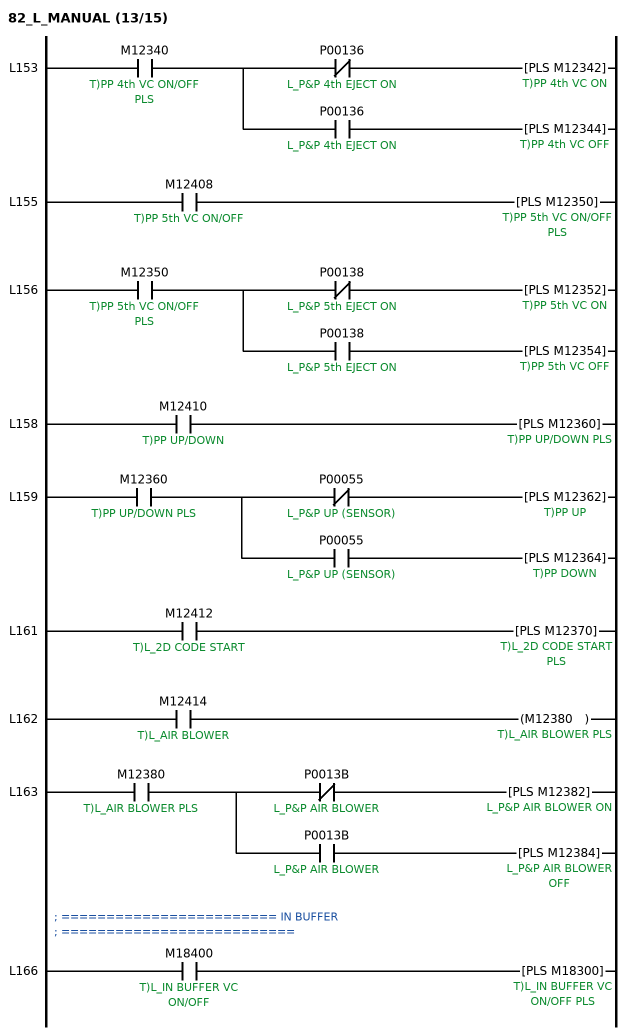
[picture p336: 82_L_MANUAL rungs L153-L166]
; L153
LOAD      M12340	// T)PP 4th VC ON/OFF PLS
MPUSH
AND NOT   P00136	// L_P&P 4th EJECT ON
OUTP      M12342	// T)PP 4th VC ON
MPOP
AND       P00136	// L_P&P 4th EJECT ON
OUTP      M12344	// T)PP 4th VC OFF
; L155
LOAD      M12408	// T)PP 5th VC ON/OFF
OUTP      M12350	// T)PP 5th VC ON/OFF PLS
; L156
LOAD      M12350	// T)PP 5th VC ON/OFF PLS
MPUSH
AND NOT   P00138	// L_P&P 5th EJECT ON
OUTP      M12352	// T)PP 5th VC ON
MPOP
AND       P00138	// L_P&P 5th EJECT ON
OUTP      M12354	// T)PP 5th VC OFF
; L158
LOAD      M12410	// T)PP UP/DOWN
OUTP      M12360	// T)PP UP/DOWN PLS
; L159
LOAD      M12360	// T)PP UP/DOWN PLS
MPUSH
AND NOT   P00055	// L_P&P UP (SENSOR)
OUTP      M12362	// T)PP UP
MPOP
AND       P00055	// L_P&P UP (SENSOR)
OUTP      M12364	// T)PP DOWN
; L161
LOAD      M12412	// T)L_2D CODE START
OUTP      M12370	// T)L_2D CODE START PLS
; L162
LOAD      M12414	// T)L_AIR BLOWER
OUT       M12380	// T)L_AIR BLOWER PLS
; L163
LOAD      M12380	// T)L_AIR BLOWER PLS
MPUSH
AND NOT   P0013B	// L_P&P AIR BLOWER
OUTP      M12382	// L_P&P AIR BLOWER ON
MPOP
AND       P0013B	// L_P&P AIR BLOWER
OUTP      M12384	// L_P&P AIR BLOWER OFF
// ======================== IN BUFFER ==========================
; L166
LOAD      M18400	// T)L_IN BUFFER VC ON/OFF
OUTP      M18300	// T)L_IN BUFFER VC ON/OFF PLS

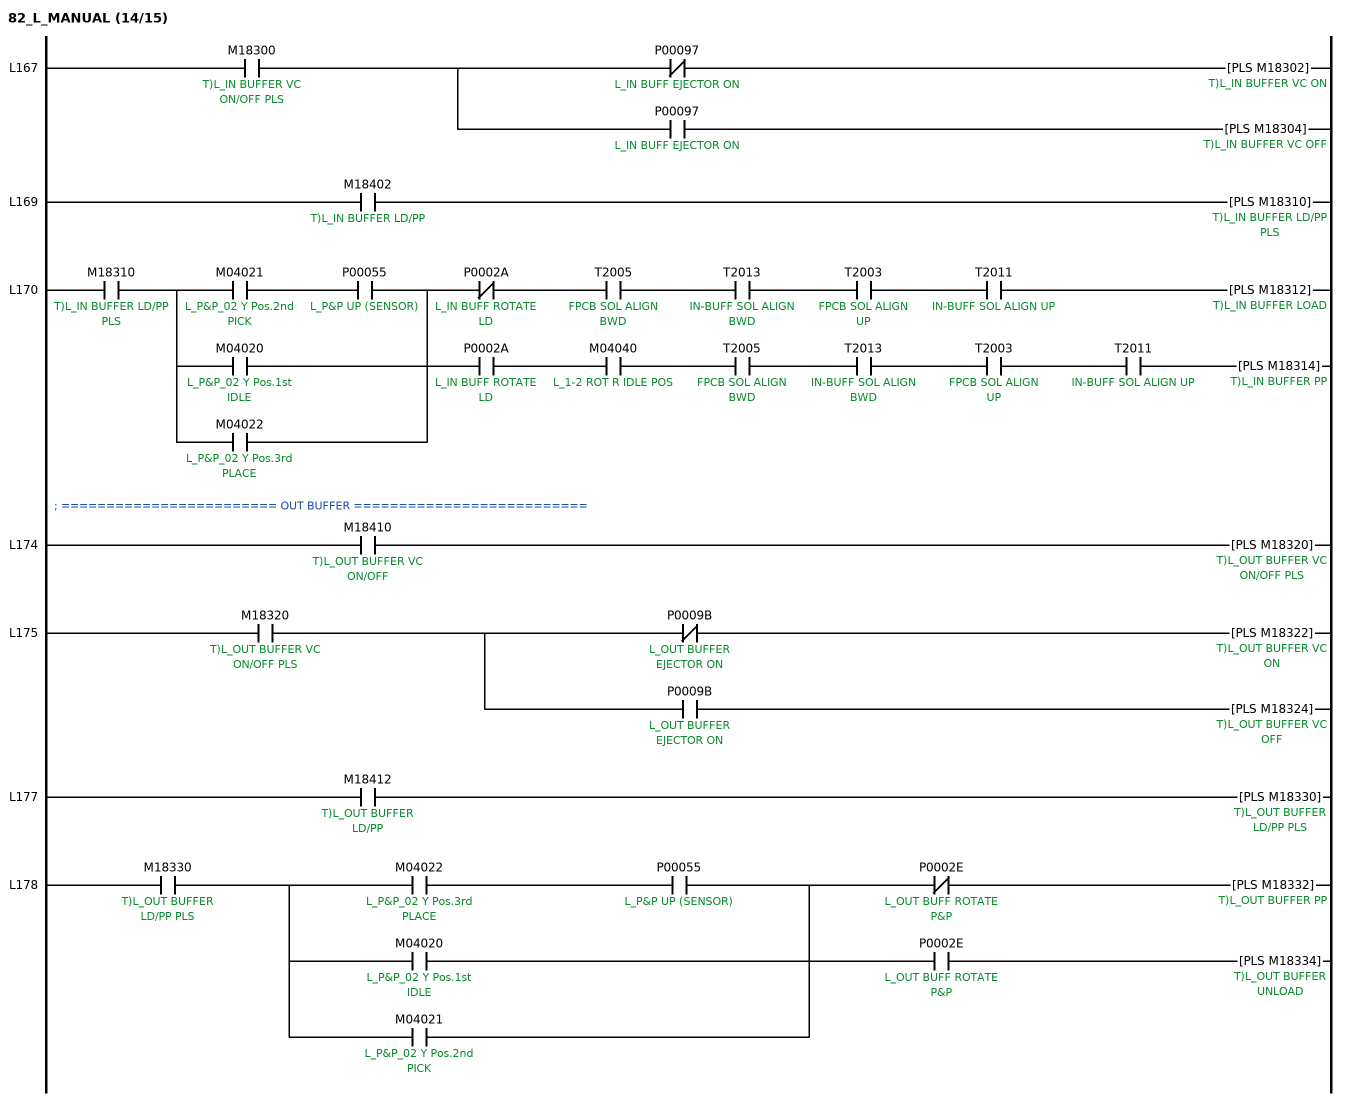
; L167
LOAD      M18300	// T)L_IN BUFFER VC ON/OFF PLS
MPUSH
AND NOT   P00097	// L_IN BUFF EJECTOR ON
OUTP      M18302	// T)L_IN BUFFER VC ON
MPOP
AND       P00097	// L_IN BUFF EJECTOR ON
OUTP      M18304	// T)L_IN BUFFER VC OFF
; L169
LOAD      M18402	// T)L_IN BUFFER LD/PP
OUTP      M18310	// T)L_IN BUFFER LD/PP PLS
; L170
LOAD      M18310	// T)L_IN BUFFER LD/PP PLS
LOAD      M04021	// L_P&P_02 Y Pos.2nd PICK
AND       P00055	// L_P&P UP (SENSOR)
OR        M04020	// L_P&P_02 Y Pos.1st IDLE
OR        M04022	// L_P&P_02 Y Pos.3rd PLACE
AND LOAD
MPUSH
AND NOT   P0002A	// L_IN BUFF ROTATE     LD
AND       T2005	// FPCB SOL ALIGN         BWD
AND       T2013	// IN-BUFF SOL ALIGN BWD
AND       T2003	// FPCB SOL ALIGN         UP
AND       T2011	// IN-BUFF SOL ALIGN UP
OUTP      M18312	// T)L_IN BUFFER LOAD
MPOP
AND       P0002A	// L_IN BUFF ROTATE     LD
AND       M04040	// L_1-2 ROT R IDLE POS
AND       T2005	// FPCB SOL ALIGN         BWD
AND       T2013	// IN-BUFF SOL ALIGN BWD
AND       T2003	// FPCB SOL ALIGN         UP
AND       T2011	// IN-BUFF SOL ALIGN UP
OUTP      M18314	// T)L_IN BUFFER PP
// ======================== OUT BUFFER ==========================
; L174
LOAD      M18410	// T)L_OUT BUFFER VC ON/OFF
OUTP      M18320	// T)L_OUT BUFFER VC ON/OFF PLS
; L175
LOAD      M18320	// T)L_OUT BUFFER VC ON/OFF PLS
MPUSH
AND NOT   P0009B	// L_OUT BUFFER EJECTOR ON
OUTP      M18322	// T)L_OUT BUFFER VC ON
MPOP
AND       P0009B	// L_OUT BUFFER EJECTOR ON
OUTP      M18324	// T)L_OUT BUFFER VC OFF
; L177
LOAD      M18412	// T)L_OUT BUFFER LD/PP
OUTP      M18330	// T)L_OUT BUFFER LD/PP PLS
; L178
LOAD      M18330	// T)L_OUT BUFFER LD/PP PLS
LOAD      M04022	// L_P&P_02 Y Pos.3rd PLACE
AND       P00055	// L_P&P UP (SENSOR)
OR        M04020	// L_P&P_02 Y Pos.1st IDLE
OR        M04021	// L_P&P_02 Y Pos.2nd PICK
AND LOAD
MPUSH
AND NOT   P0002E	// L_OUT BUFF ROTATE      P&P
OUTP      M18332	// T)L_OUT BUFFER PP
MPOP
AND       P0002E	// L_OUT BUFF ROTATE      P&P
OUTP      M18334	// T)L_OUT BUFFER UNLOAD

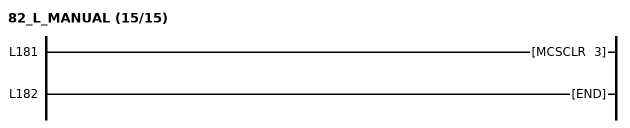
; L181
MCSCLR    3
; L182
END

PROGRAM 83_R_MANUAL (task: ¨ö¨¬A¥ì CA¡¤I¡¾¡¿¡¤¡Í)

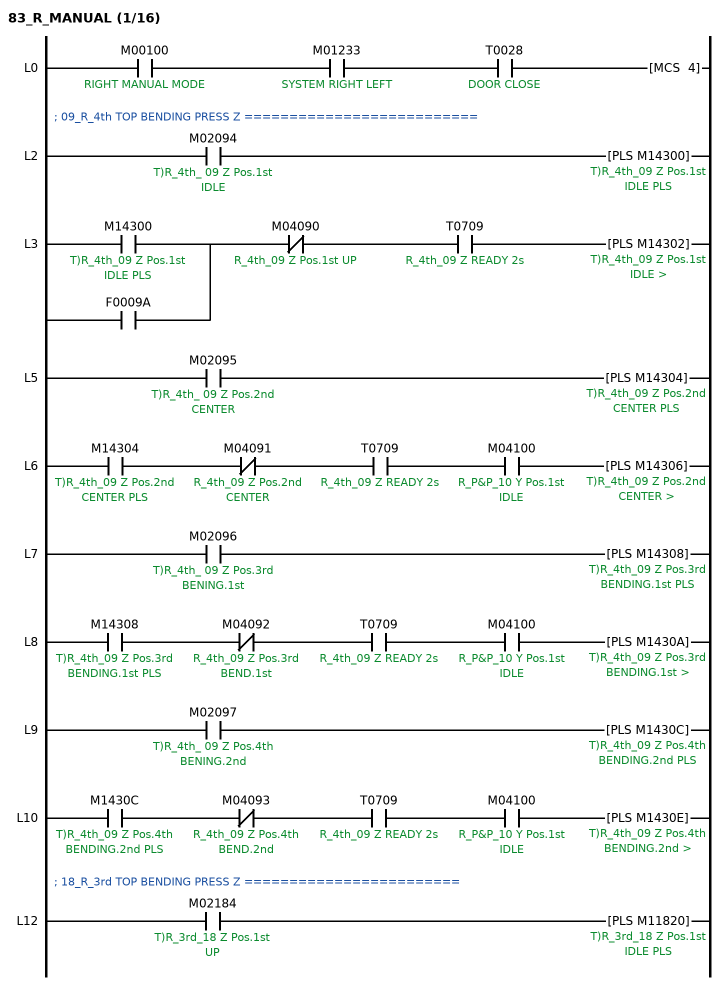
; L0
LOAD      M00100	// RIGHT MANUAL MODE
AND       M01233	// SYSTEM RIGHT LEFT
AND       T0028	// DOOR CLOSE
MCS       4
// 09_R_4th TOP BENDING PRESS Z ==========================
; L2
LOAD      M02094	// T)R_4th_ 09 Z Pos.1st IDLE
OUTP      M14300	// T)R_4th_09 Z Pos.1st IDLE PLS
; L3
LOAD      M14300	// T)R_4th_09 Z Pos.1st IDLE PLS
OR        F0009A
AND NOT   M04090	// R_4th_09 Z Pos.1st UP
AND       T0709	// R_4th_09 Z READY 2s
OUTP      M14302	// T)R_4th_09 Z Pos.1st IDLE >
; L5
LOAD      M02095	// T)R_4th_ 09 Z Pos.2nd CENTER
OUTP      M14304	// T)R_4th_09 Z Pos.2nd CENTER PLS
; L6
LOAD      M14304	// T)R_4th_09 Z Pos.2nd CENTER PLS
AND NOT   M04091	// R_4th_09 Z Pos.2nd CENTER
AND       T0709	// R_4th_09 Z READY 2s
AND       M04100	// R_P&P_10 Y Pos.1st IDLE
OUTP      M14306	// T)R_4th_09 Z Pos.2nd CENTER >
; L7
LOAD      M02096	// T)R_4th_ 09 Z Pos.3rd BENING.1st
OUTP      M14308	// T)R_4th_09 Z Pos.3rd BENDING.1st PLS
; L8
LOAD      M14308	// T)R_4th_09 Z Pos.3rd BENDING.1st PLS
AND NOT   M04092	// R_4th_09 Z Pos.3rd BEND.1st
AND       T0709	// R_4th_09 Z READY 2s
AND       M04100	// R_P&P_10 Y Pos.1st IDLE
OUTP      M1430A	// T)R_4th_09 Z Pos.3rd BENDING.1st >
; L9
LOAD      M02097	// T)R_4th_ 09 Z Pos.4th BENING.2nd
OUTP      M1430C	// T)R_4th_09 Z Pos.4th BENDING.2nd PLS
; L10
LOAD      M1430C	// T)R_4th_09 Z Pos.4th BENDING.2nd PLS
AND NOT   M04093	// R_4th_09 Z Pos.4th BEND.2nd
AND       T0709	// R_4th_09 Z READY 2s
AND       M04100	// R_P&P_10 Y Pos.1st IDLE
OUTP      M1430E	// T)R_4th_09 Z Pos.4th BENDING.2nd >
// 18_R_3rd TOP BENDING PRESS Z ======================== 
; L12
LOAD      M02184	// T)R_3rd_18 Z Pos.1st UP
OUTP      M11820	// T)R_3rd_18 Z Pos.1st IDLE PLS

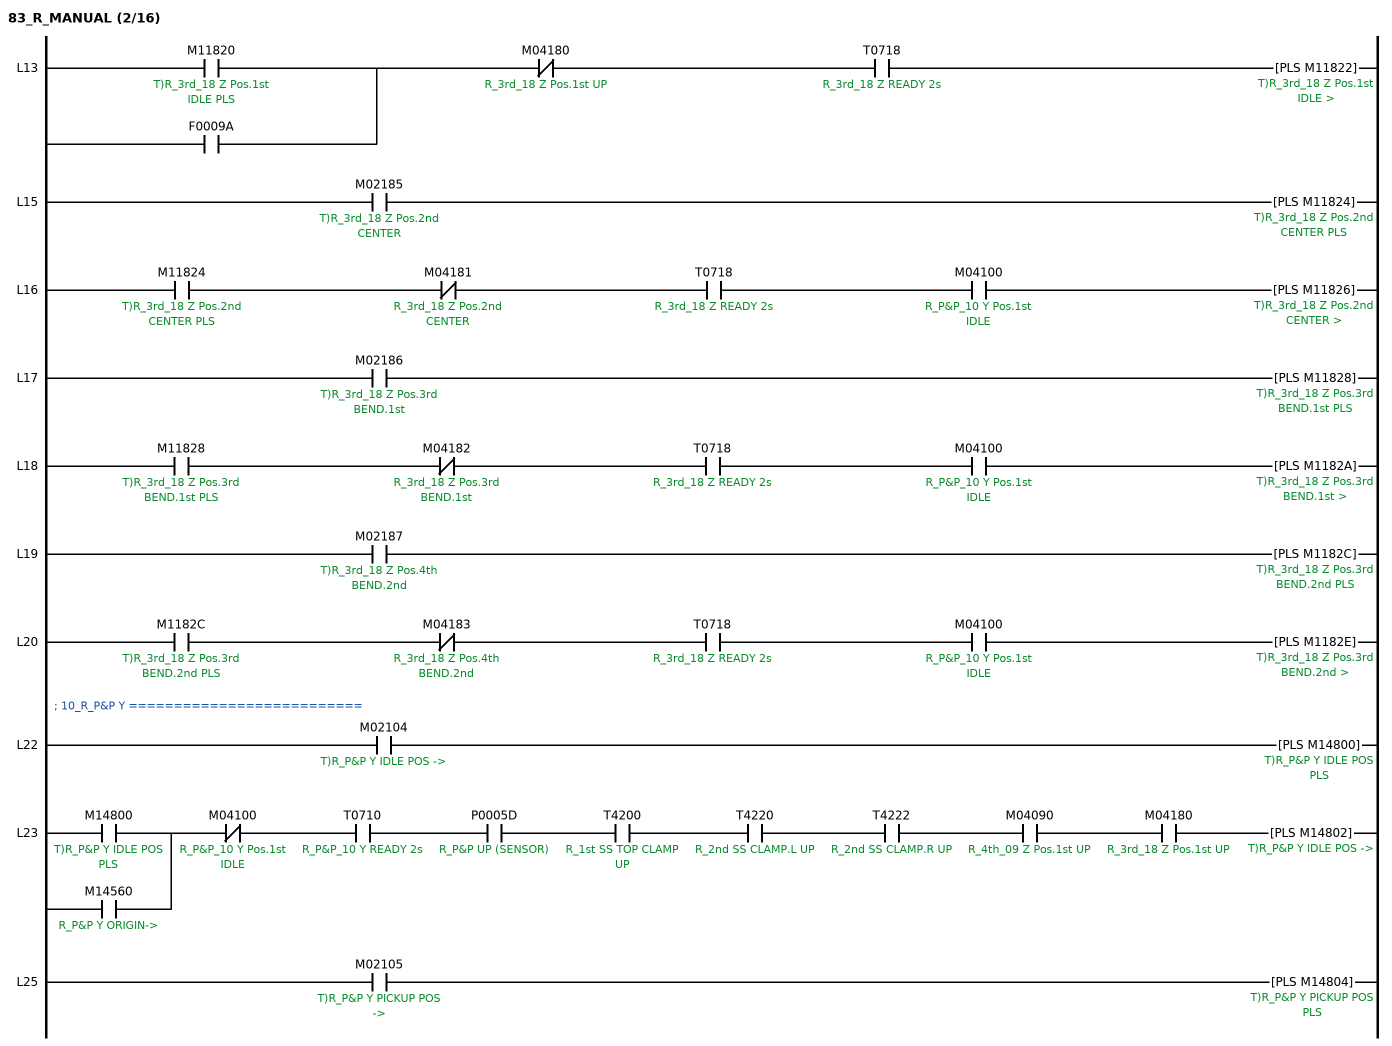
; L13
LOAD      M11820	// T)R_3rd_18 Z Pos.1st IDLE PLS
OR        F0009A
AND NOT   M04180	// R_3rd_18 Z Pos.1st UP
AND       T0718	// R_3rd_18 Z READY 2s
OUTP      M11822	// T)R_3rd_18 Z Pos.1st IDLE >
; L15
LOAD      M02185	// T)R_3rd_18 Z Pos.2nd CENTER
OUTP      M11824	// T)R_3rd_18 Z Pos.2nd CENTER PLS
; L16
LOAD      M11824	// T)R_3rd_18 Z Pos.2nd CENTER PLS
AND NOT   M04181	// R_3rd_18 Z Pos.2nd CENTER
AND       T0718	// R_3rd_18 Z READY 2s
AND       M04100	// R_P&P_10 Y Pos.1st IDLE
OUTP      M11826	// T)R_3rd_18 Z Pos.2nd CENTER >
; L17
LOAD      M02186	// T)R_3rd_18 Z Pos.3rd BEND.1st
OUTP      M11828	// T)R_3rd_18 Z Pos.3rd BEND.1st PLS
; L18
LOAD      M11828	// T)R_3rd_18 Z Pos.3rd BEND.1st PLS
AND NOT   M04182	// R_3rd_18 Z Pos.3rd BEND.1st
AND       T0718	// R_3rd_18 Z READY 2s
AND       M04100	// R_P&P_10 Y Pos.1st IDLE
OUTP      M1182A	// T)R_3rd_18 Z Pos.3rd BEND.1st >
; L19
LOAD      M02187	// T)R_3rd_18 Z Pos.4th BEND.2nd
OUTP      M1182C	// T)R_3rd_18 Z Pos.3rd BEND.2nd PLS
; L20
LOAD      M1182C	// T)R_3rd_18 Z Pos.3rd BEND.2nd PLS
AND NOT   M04183	// R_3rd_18 Z Pos.4th BEND.2nd
AND       T0718	// R_3rd_18 Z READY 2s
AND       M04100	// R_P&P_10 Y Pos.1st IDLE
OUTP      M1182E	// T)R_3rd_18 Z Pos.3rd BEND.2nd >
// 10_R_P&P Y ==========================
; L22
LOAD      M02104	// T)R_P&P Y IDLE POS ->
OUTP      M14800	// T)R_P&P Y IDLE POS PLS
; L23
LOAD      M14800	// T)R_P&P Y IDLE POS PLS
OR        M14560	// R_P&P Y ORIGIN->
AND NOT   M04100	// R_P&P_10 Y Pos.1st IDLE
AND       T0710	// R_P&P_10 Y READY 2s
AND       P0005D	// R_P&P UP (SENSOR)
AND       T4200	// R_1st SS TOP CLAMP UP
AND       T4220	// R_2nd SS CLAMP.L UP
AND       T4222	// R_2nd SS CLAMP.R UP
AND       M04090	// R_4th_09 Z Pos.1st UP
AND       M04180	// R_3rd_18 Z Pos.1st UP
OUTP      M14802	// T)R_P&P Y IDLE POS ->
; L25
LOAD      M02105	// T)R_P&P Y PICKUP POS ->
OUTP      M14804	// T)R_P&P Y PICKUP POS PLS

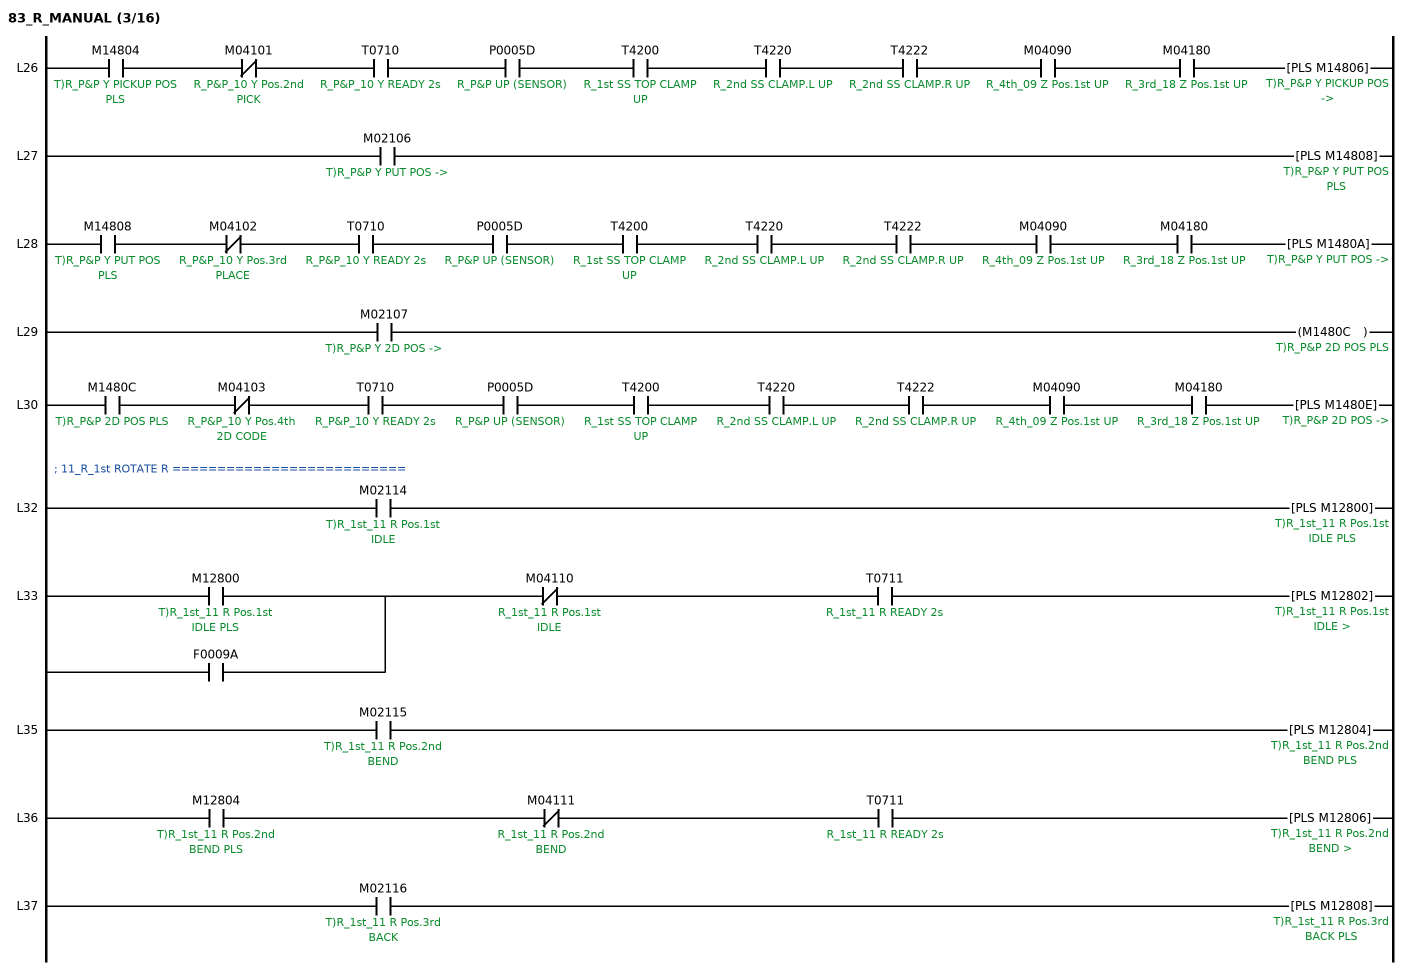
; L26
LOAD      M14804	// T)R_P&P Y PICKUP POS PLS
AND NOT   M04101	// R_P&P_10 Y Pos.2nd PICK
AND       T0710	// R_P&P_10 Y READY 2s
AND       P0005D	// R_P&P UP (SENSOR)
AND       T4200	// R_1st SS TOP CLAMP UP
AND       T4220	// R_2nd SS CLAMP.L UP
AND       T4222	// R_2nd SS CLAMP.R UP
AND       M04090	// R_4th_09 Z Pos.1st UP
AND       M04180	// R_3rd_18 Z Pos.1st UP
OUTP      M14806	// T)R_P&P Y PICKUP POS ->
; L27
LOAD      M02106	// T)R_P&P Y PUT POS ->
OUTP      M14808	// T)R_P&P Y PUT POS PLS
; L28
LOAD      M14808	// T)R_P&P Y PUT POS PLS
AND NOT   M04102	// R_P&P_10 Y Pos.3rd PLACE
AND       T0710	// R_P&P_10 Y READY 2s
AND       P0005D	// R_P&P UP (SENSOR)
AND       T4200	// R_1st SS TOP CLAMP UP
AND       T4220	// R_2nd SS CLAMP.L UP
AND       T4222	// R_2nd SS CLAMP.R UP
AND       M04090	// R_4th_09 Z Pos.1st UP
AND       M04180	// R_3rd_18 Z Pos.1st UP
OUTP      M1480A	// T)R_P&P Y PUT POS ->
; L29
LOAD      M02107	// T)R_P&P Y 2D POS ->
OUT       M1480C	// T)R_P&P 2D POS PLS
; L30
LOAD      M1480C	// T)R_P&P 2D POS PLS
AND NOT   M04103	// R_P&P_10 Y Pos.4th 2D CODE
AND       T0710	// R_P&P_10 Y READY 2s
AND       P0005D	// R_P&P UP (SENSOR)
AND       T4200	// R_1st SS TOP CLAMP UP
AND       T4220	// R_2nd SS CLAMP.L UP
AND       T4222	// R_2nd SS CLAMP.R UP
AND       M04090	// R_4th_09 Z Pos.1st UP
AND       M04180	// R_3rd_18 Z Pos.1st UP
OUTP      M1480E	// T)R_P&P 2D POS ->
// 11_R_1st ROTATE R ==========================
; L32
LOAD      M02114	// T)R_1st_11 R Pos.1st IDLE
OUTP      M12800	// T)R_1st_11 R Pos.1st IDLE PLS
; L33
LOAD      M12800	// T)R_1st_11 R Pos.1st IDLE PLS
OR        F0009A
AND NOT   M04110	// R_1st_11 R Pos.1st IDLE
AND       T0711	// R_1st_11 R READY 2s
OUTP      M12802	// T)R_1st_11 R Pos.1st IDLE >
; L35
LOAD      M02115	// T)R_1st_11 R Pos.2nd BEND
OUTP      M12804	// T)R_1st_11 R Pos.2nd BEND PLS
; L36
LOAD      M12804	// T)R_1st_11 R Pos.2nd BEND PLS
AND NOT   M04111	// R_1st_11 R Pos.2nd BEND
AND       T0711	// R_1st_11 R READY 2s
OUTP      M12806	// T)R_1st_11 R Pos.2nd BEND >
; L37
LOAD      M02116	// T)R_1st_11 R Pos.3rd BACK
OUTP      M12808	// T)R_1st_11 R Pos.3rd BACK PLS

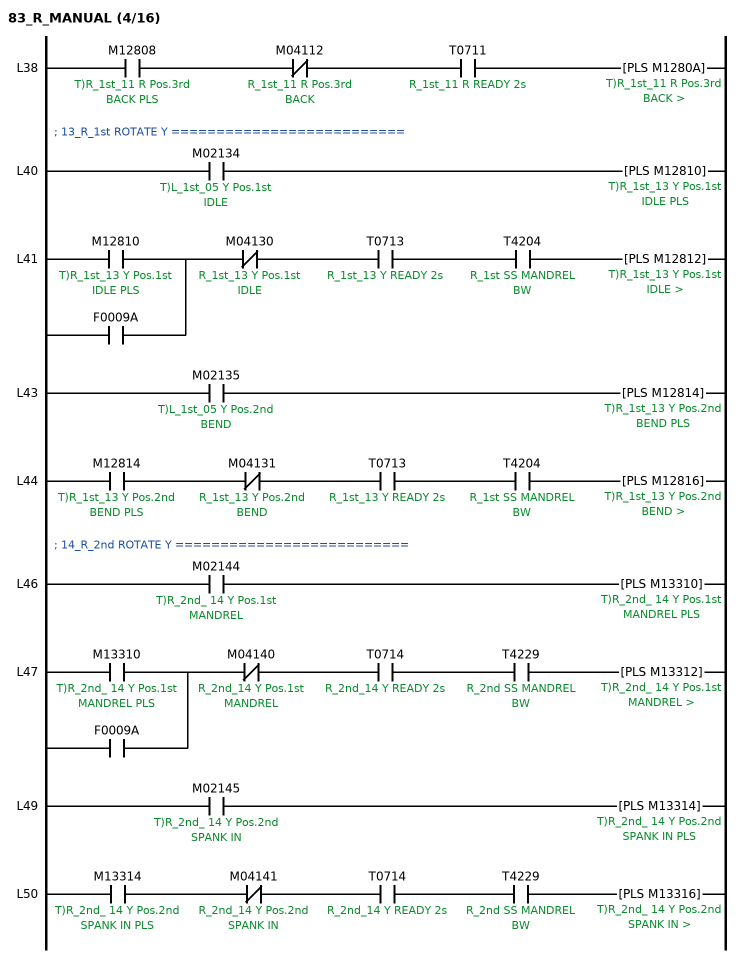
; L38
LOAD      M12808	// T)R_1st_11 R Pos.3rd BACK PLS
AND NOT   M04112	// R_1st_11 R Pos.3rd BACK
AND       T0711	// R_1st_11 R READY 2s
OUTP      M1280A	// T)R_1st_11 R Pos.3rd BACK >
// 13_R_1st ROTATE Y ==========================
; L40
LOAD      M02134	// T)L_1st_05 Y Pos.1st IDLE
OUTP      M12810	// T)R_1st_13 Y Pos.1st IDLE PLS
; L41
LOAD      M12810	// T)R_1st_13 Y Pos.1st IDLE PLS
OR        F0009A
AND NOT   M04130	// R_1st_13 Y Pos.1st IDLE
AND       T0713	// R_1st_13 Y READY 2s
AND       T4204	// R_1st SS MANDREL BW
OUTP      M12812	// T)R_1st_13 Y Pos.1st IDLE >
; L43
LOAD      M02135	// T)L_1st_05 Y Pos.2nd BEND
OUTP      M12814	// T)R_1st_13 Y Pos.2nd BEND PLS
; L44
LOAD      M12814	// T)R_1st_13 Y Pos.2nd BEND PLS
AND NOT   M04131	// R_1st_13 Y Pos.2nd BEND
AND       T0713	// R_1st_13 Y READY 2s
AND       T4204	// R_1st SS MANDREL BW
OUTP      M12816	// T)R_1st_13 Y Pos.2nd BEND >
// 14_R_2nd ROTATE Y ==========================
; L46
LOAD      M02144	// T)R_2nd_ 14 Y Pos.1st MANDREL
OUTP      M13310	// T)R_2nd_ 14 Y Pos.1st MANDREL PLS
; L47
LOAD      M13310	// T)R_2nd_ 14 Y Pos.1st MANDREL PLS
OR        F0009A
AND NOT   M04140	// R_2nd_14 Y Pos.1st MANDREL
AND       T0714	// R_2nd_14 Y READY 2s
AND       T4229	// R_2nd SS MANDREL BW
OUTP      M13312	// T)R_2nd_ 14 Y Pos.1st MANDREL >
; L49
LOAD      M02145	// T)R_2nd_ 14 Y Pos.2nd SPANK IN
OUTP      M13314	// T)R_2nd_ 14 Y Pos.2nd SPANK IN PLS
; L50
LOAD      M13314	// T)R_2nd_ 14 Y Pos.2nd SPANK IN PLS
AND NOT   M04141	// R_2nd_14 Y Pos.2nd SPANK IN
AND       T0714	// R_2nd_14 Y READY 2s
AND       T4229	// R_2nd SS MANDREL BW
OUTP      M13316	// T)R_2nd_ 14 Y Pos.2nd SPANK IN >

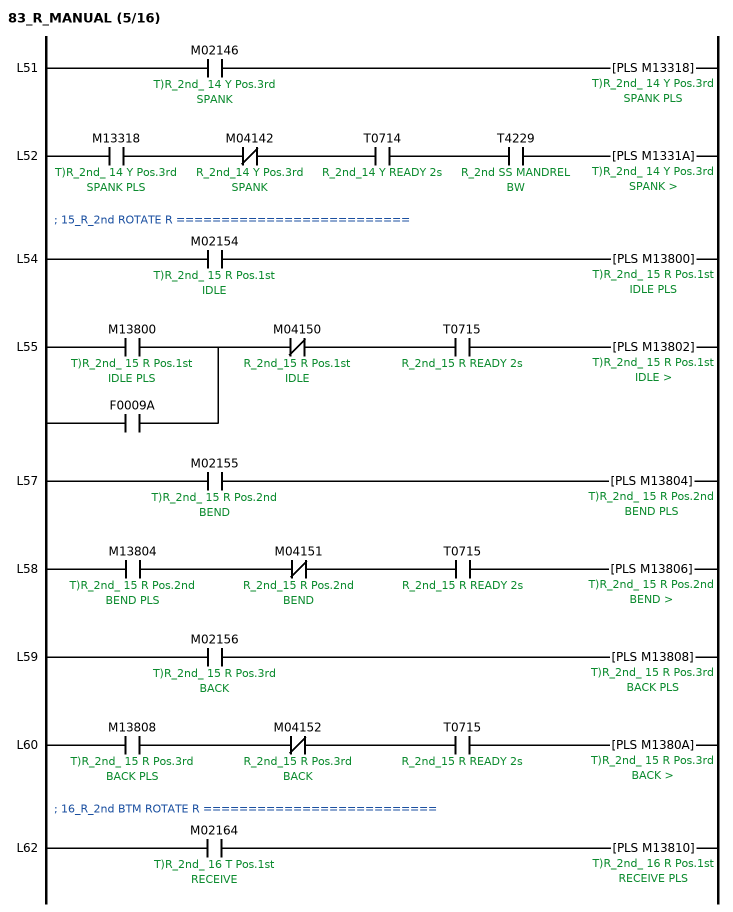
; L51
LOAD      M02146	// T)R_2nd_ 14 Y Pos.3rd SPANK
OUTP      M13318	// T)R_2nd_ 14 Y Pos.3rd SPANK PLS
; L52
LOAD      M13318	// T)R_2nd_ 14 Y Pos.3rd SPANK PLS
AND NOT   M04142	// R_2nd_14 Y Pos.3rd SPANK
AND       T0714	// R_2nd_14 Y READY 2s
AND       T4229	// R_2nd SS MANDREL BW
OUTP      M1331A	// T)R_2nd_ 14 Y Pos.3rd SPANK >
// 15_R_2nd ROTATE R ==========================
; L54
LOAD      M02154	// T)R_2nd_ 15 R Pos.1st IDLE
OUTP      M13800	// T)R_2nd_ 15 R Pos.1st IDLE PLS
; L55
LOAD      M13800	// T)R_2nd_ 15 R Pos.1st IDLE PLS
OR        F0009A
AND NOT   M04150	// R_2nd_15 R Pos.1st IDLE
AND       T0715	// R_2nd_15 R READY 2s
OUTP      M13802	// T)R_2nd_ 15 R Pos.1st IDLE >
; L57
LOAD      M02155	// T)R_2nd_ 15 R Pos.2nd BEND
OUTP      M13804	// T)R_2nd_ 15 R Pos.2nd BEND PLS
; L58
LOAD      M13804	// T)R_2nd_ 15 R Pos.2nd BEND PLS
AND NOT   M04151	// R_2nd_15 R Pos.2nd BEND
AND       T0715	// R_2nd_15 R READY 2s
OUTP      M13806	// T)R_2nd_ 15 R Pos.2nd BEND >
; L59
LOAD      M02156	// T)R_2nd_ 15 R Pos.3rd BACK
OUTP      M13808	// T)R_2nd_ 15 R Pos.3rd BACK PLS
; L60
LOAD      M13808	// T)R_2nd_ 15 R Pos.3rd BACK PLS
AND NOT   M04152	// R_2nd_15 R Pos.3rd BACK
AND       T0715	// R_2nd_15 R READY 2s
OUTP      M1380A	// T)R_2nd_ 15 R Pos.3rd BACK >
// 16_R_2nd BTM ROTATE R ==========================
; L62
LOAD      M02164	// T)R_2nd_ 16 T Pos.1st RECEIVE
OUTP      M13810	// T)R_2nd_ 16 R Pos.1st RECEIVE PLS

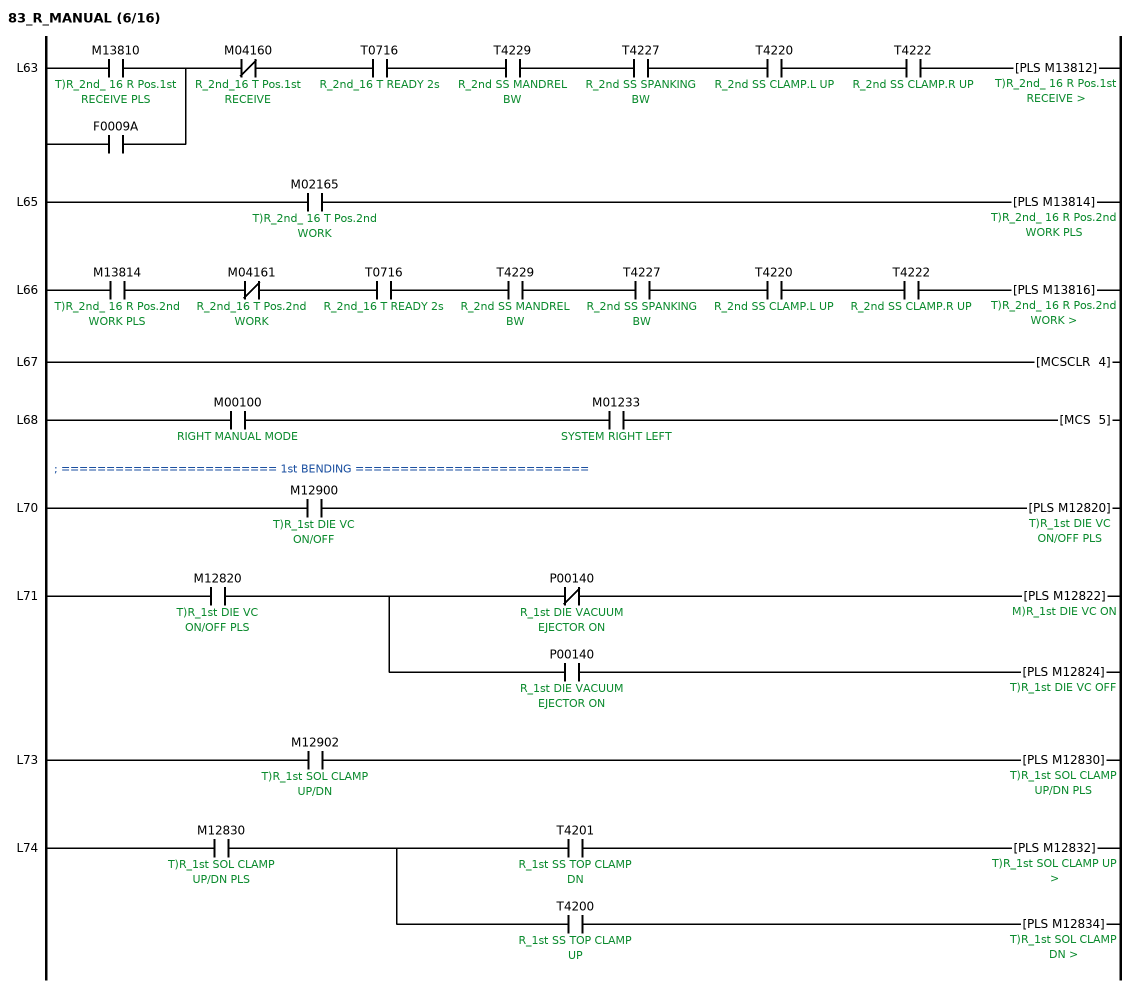
; L63
LOAD      M13810	// T)R_2nd_ 16 R Pos.1st RECEIVE PLS
OR        F0009A
AND NOT   M04160	// R_2nd_16 T Pos.1st RECEIVE
AND       T0716	// R_2nd_16 T READY 2s
AND       T4229	// R_2nd SS MANDREL BW
AND       T4227	// R_2nd SS SPANKING BW
AND       T4220	// R_2nd SS CLAMP.L UP
AND       T4222	// R_2nd SS CLAMP.R UP
OUTP      M13812	// T)R_2nd_ 16 R Pos.1st RECEIVE >
; L65
LOAD      M02165	// T)R_2nd_ 16 T Pos.2nd WORK
OUTP      M13814	// T)R_2nd_ 16 R Pos.2nd WORK PLS
; L66
LOAD      M13814	// T)R_2nd_ 16 R Pos.2nd WORK PLS
AND NOT   M04161	// R_2nd_16 T Pos.2nd WORK
AND       T0716	// R_2nd_16 T READY 2s
AND       T4229	// R_2nd SS MANDREL BW
AND       T4227	// R_2nd SS SPANKING BW
AND       T4220	// R_2nd SS CLAMP.L UP
AND       T4222	// R_2nd SS CLAMP.R UP
OUTP      M13816	// T)R_2nd_ 16 R Pos.2nd WORK >
; L67
MCSCLR    4
; L68
LOAD      M00100	// RIGHT MANUAL MODE
AND       M01233	// SYSTEM RIGHT LEFT
MCS       5
// ======================== 1st BENDING ==========================
; L70
LOAD      M12900	// T)R_1st DIE VC ON/OFF
OUTP      M12820	// T)R_1st DIE VC ON/OFF PLS
; L71
LOAD      M12820	// T)R_1st DIE VC ON/OFF PLS
MPUSH
AND NOT   P00140	// R_1st DIE VACUUM EJECTOR ON
OUTP      M12822	// M)R_1st DIE VC ON
MPOP
AND       P00140	// R_1st DIE VACUUM EJECTOR ON
OUTP      M12824	// T)R_1st DIE VC OFF
; L73
LOAD      M12902	// T)R_1st SOL CLAMP UP/DN
OUTP      M12830	// T)R_1st SOL CLAMP UP/DN PLS
; L74
LOAD      M12830	// T)R_1st SOL CLAMP UP/DN PLS
MPUSH
AND       T4201	// R_1st SS TOP CLAMP DN
OUTP      M12832	// T)R_1st SOL CLAMP UP >
MPOP
AND       T4200	// R_1st SS TOP CLAMP UP
OUTP      M12834	// T)R_1st SOL CLAMP DN >

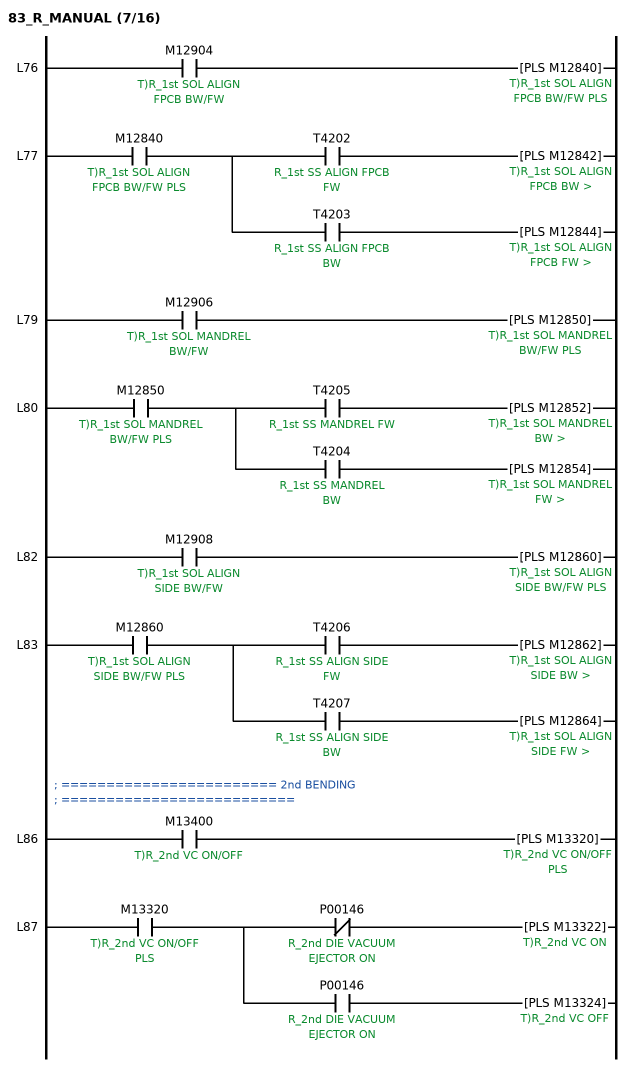
; L76
LOAD      M12904	// T)R_1st SOL ALIGN FPCB BW/FW
OUTP      M12840	// T)R_1st SOL ALIGN FPCB BW/FW PLS
; L77
LOAD      M12840	// T)R_1st SOL ALIGN FPCB BW/FW PLS
MPUSH
AND       T4202	// R_1st SS ALIGN FPCB FW
OUTP      M12842	// T)R_1st SOL ALIGN FPCB BW >
MPOP
AND       T4203	// R_1st SS ALIGN FPCB BW
OUTP      M12844	// T)R_1st SOL ALIGN FPCB FW >
; L79
LOAD      M12906	// T)R_1st SOL MANDREL BW/FW
OUTP      M12850	// T)R_1st SOL MANDREL BW/FW PLS
; L80
LOAD      M12850	// T)R_1st SOL MANDREL BW/FW PLS
MPUSH
AND       T4205	// R_1st SS MANDREL FW
OUTP      M12852	// T)R_1st SOL MANDREL BW >
MPOP
AND       T4204	// R_1st SS MANDREL BW
OUTP      M12854	// T)R_1st SOL MANDREL FW >
; L82
LOAD      M12908	// T)R_1st SOL ALIGN SIDE BW/FW
OUTP      M12860	// T)R_1st SOL ALIGN SIDE BW/FW PLS
; L83
LOAD      M12860	// T)R_1st SOL ALIGN SIDE BW/FW PLS
MPUSH
AND       T4206	// R_1st SS ALIGN SIDE FW
OUTP      M12862	// T)R_1st SOL ALIGN SIDE BW >
MPOP
AND       T4207	// R_1st SS ALIGN SIDE BW
OUTP      M12864	// T)R_1st SOL ALIGN SIDE FW >
// ======================== 2nd BENDING ==========================
; L86
LOAD      M13400	// T)R_2nd VC ON/OFF
OUTP      M13320	// T)R_2nd VC ON/OFF PLS
; L87
LOAD      M13320	// T)R_2nd VC ON/OFF PLS
MPUSH
AND NOT   P00146	// R_2nd DIE VACUUM EJECTOR ON
OUTP      M13322	// T)R_2nd VC ON
MPOP
AND       P00146	// R_2nd DIE VACUUM EJECTOR ON
OUTP      M13324	// T)R_2nd VC OFF

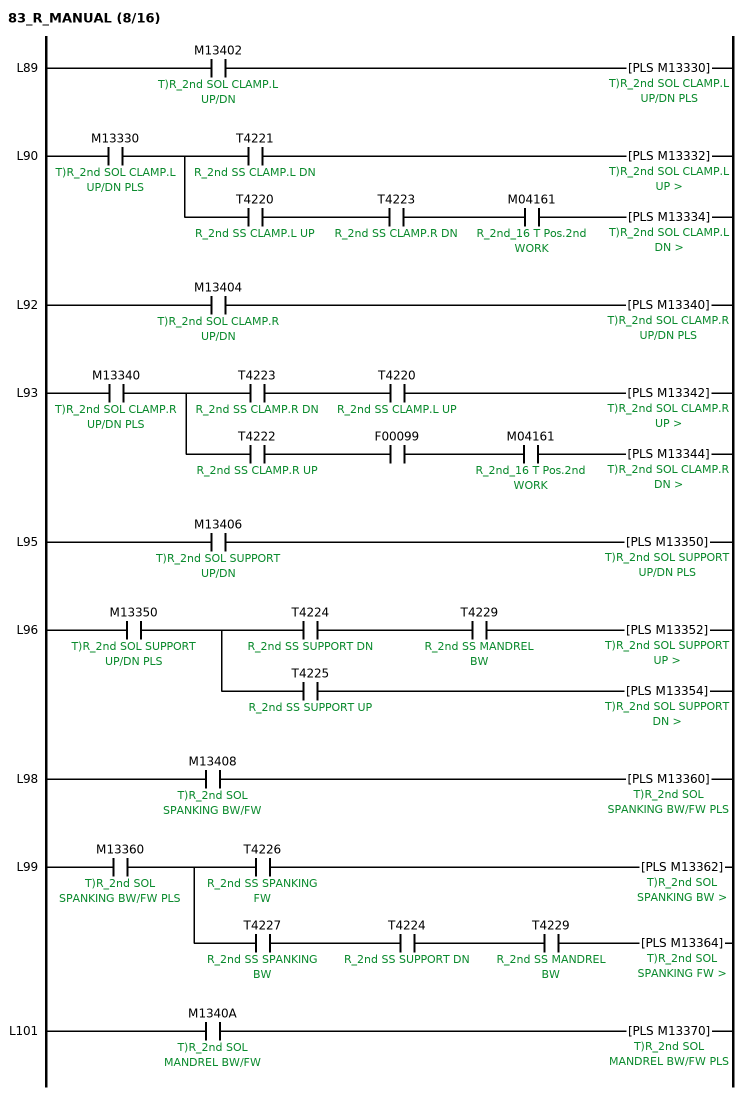
; L89
LOAD      M13402	// T)R_2nd SOL CLAMP.L UP/DN
OUTP      M13330	// T)R_2nd SOL CLAMP.L UP/DN PLS
; L90
LOAD      M13330	// T)R_2nd SOL CLAMP.L UP/DN PLS
MPUSH
AND       T4221	// R_2nd SS CLAMP.L DN
OUTP      M13332	// T)R_2nd SOL CLAMP.L UP >
MPOP
AND       T4220	// R_2nd SS CLAMP.L UP
AND       T4223	// R_2nd SS CLAMP.R DN
AND       M04161	// R_2nd_16 T Pos.2nd WORK
OUTP      M13334	// T)R_2nd SOL CLAMP.L DN >
; L92
LOAD      M13404	// T)R_2nd SOL CLAMP.R UP/DN
OUTP      M13340	// T)R_2nd SOL CLAMP.R UP/DN PLS
; L93
LOAD      M13340	// T)R_2nd SOL CLAMP.R UP/DN PLS
MPUSH
AND       T4223	// R_2nd SS CLAMP.R DN
AND       T4220	// R_2nd SS CLAMP.L UP
OUTP      M13342	// T)R_2nd SOL CLAMP.R UP >
MPOP
AND       T4222	// R_2nd SS CLAMP.R UP
AND       F00099
AND       M04161	// R_2nd_16 T Pos.2nd WORK
OUTP      M13344	// T)R_2nd SOL CLAMP.R DN >
; L95
LOAD      M13406	// T)R_2nd SOL SUPPORT UP/DN
OUTP      M13350	// T)R_2nd SOL SUPPORT UP/DN PLS
; L96
LOAD      M13350	// T)R_2nd SOL SUPPORT UP/DN PLS
MPUSH
AND       T4224	// R_2nd SS SUPPORT DN
AND       T4229	// R_2nd SS MANDREL BW
OUTP      M13352	// T)R_2nd SOL SUPPORT UP >
MPOP
AND       T4225	// R_2nd SS SUPPORT UP
OUTP      M13354	// T)R_2nd SOL SUPPORT DN >
; L98
LOAD      M13408	// T)R_2nd SOL SPANKING BW/FW
OUTP      M13360	// T)R_2nd SOL SPANKING BW/FW PLS
; L99
LOAD      M13360	// T)R_2nd SOL SPANKING BW/FW PLS
MPUSH
AND       T4226	// R_2nd SS SPANKING FW
OUTP      M13362	// T)R_2nd SOL SPANKING BW >
MPOP
AND       T4227	// R_2nd SS SPANKING BW
AND       T4224	// R_2nd SS SUPPORT DN
AND       T4229	// R_2nd SS MANDREL BW
OUTP      M13364	// T)R_2nd SOL SPANKING FW >
; L101
LOAD      M1340A	// T)R_2nd SOL MANDREL BW/FW
OUTP      M13370	// T)R_2nd SOL MANDREL BW/FW PLS

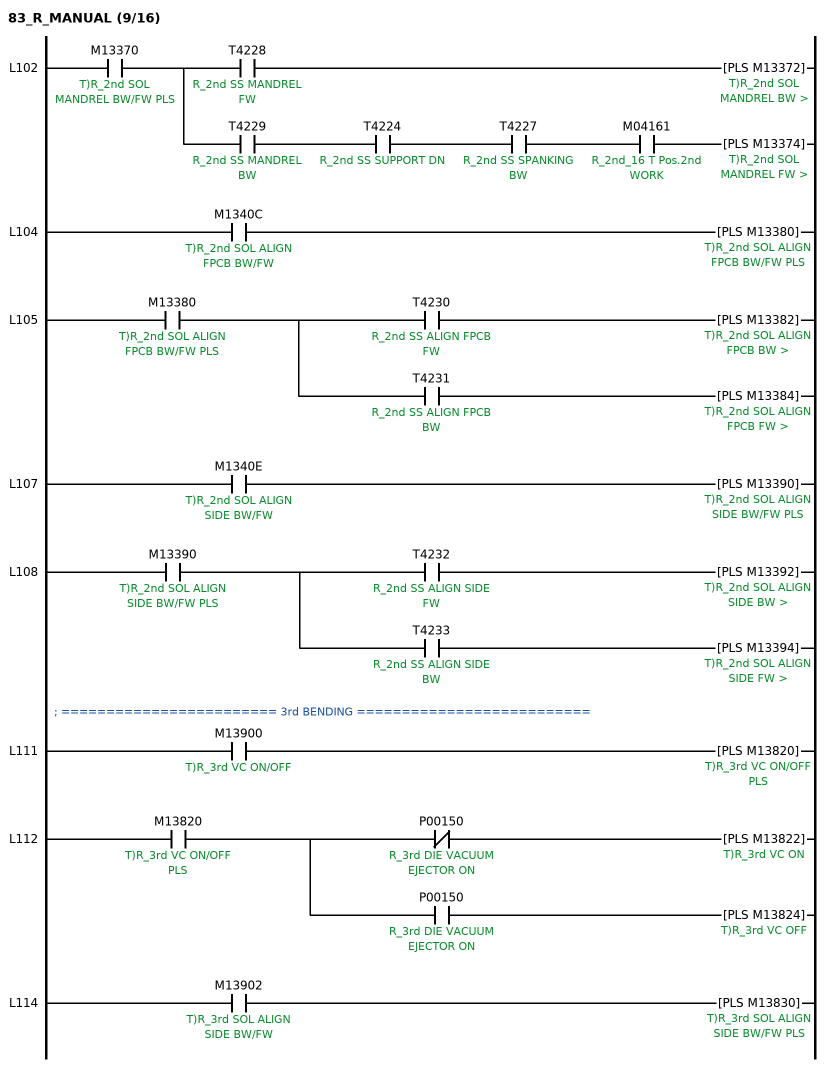
; L102
LOAD      M13370	// T)R_2nd SOL MANDREL BW/FW PLS
MPUSH
AND       T4228	// R_2nd SS MANDREL FW
OUTP      M13372	// T)R_2nd SOL MANDREL BW >
MPOP
AND       T4229	// R_2nd SS MANDREL BW
AND       T4224	// R_2nd SS SUPPORT DN
AND       T4227	// R_2nd SS SPANKING BW
AND       M04161	// R_2nd_16 T Pos.2nd WORK
OUTP      M13374	// T)R_2nd SOL MANDREL FW >
; L104
LOAD      M1340C	// T)R_2nd SOL ALIGN FPCB BW/FW
OUTP      M13380	// T)R_2nd SOL ALIGN FPCB BW/FW PLS
; L105
LOAD      M13380	// T)R_2nd SOL ALIGN FPCB BW/FW PLS
MPUSH
AND       T4230	// R_2nd SS ALIGN FPCB FW
OUTP      M13382	// T)R_2nd SOL ALIGN FPCB BW >
MPOP
AND       T4231	// R_2nd SS ALIGN FPCB BW
OUTP      M13384	// T)R_2nd SOL ALIGN FPCB FW >
; L107
LOAD      M1340E	// T)R_2nd SOL ALIGN SIDE BW/FW
OUTP      M13390	// T)R_2nd SOL ALIGN SIDE BW/FW PLS
; L108
LOAD      M13390	// T)R_2nd SOL ALIGN SIDE BW/FW PLS
MPUSH
AND       T4232	// R_2nd SS ALIGN SIDE FW
OUTP      M13392	// T)R_2nd SOL ALIGN SIDE BW >
MPOP
AND       T4233	// R_2nd SS ALIGN SIDE BW
OUTP      M13394	// T)R_2nd SOL ALIGN SIDE FW >
// ======================== 3rd BENDING ==========================
; L111
LOAD      M13900	// T)R_3rd VC ON/OFF
OUTP      M13820	// T)R_3rd VC ON/OFF PLS
; L112
LOAD      M13820	// T)R_3rd VC ON/OFF PLS
MPUSH
AND NOT   P00150	// R_3rd DIE VACUUM EJECTOR ON
OUTP      M13822	// T)R_3rd VC ON
MPOP
AND       P00150	// R_3rd DIE VACUUM EJECTOR ON
OUTP      M13824	// T)R_3rd VC OFF
; L114
LOAD      M13902	// T)R_3rd SOL ALIGN SIDE BW/FW
OUTP      M13830	// T)R_3rd SOL ALIGN SIDE BW/FW PLS

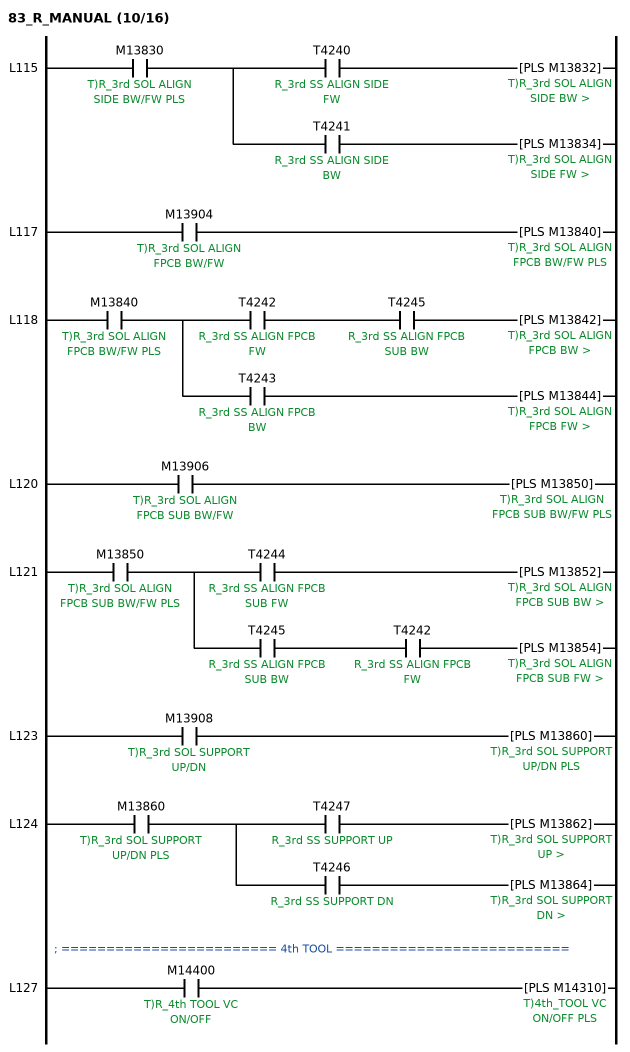
; L115
LOAD      M13830	// T)R_3rd SOL ALIGN SIDE BW/FW PLS
MPUSH
AND       T4240	// R_3rd SS ALIGN SIDE FW
OUTP      M13832	// T)R_3rd SOL ALIGN SIDE BW >
MPOP
AND       T4241	// R_3rd SS ALIGN SIDE BW
OUTP      M13834	// T)R_3rd SOL ALIGN SIDE FW >
; L117
LOAD      M13904	// T)R_3rd SOL ALIGN FPCB BW/FW
OUTP      M13840	// T)R_3rd SOL ALIGN FPCB BW/FW PLS
; L118
LOAD      M13840	// T)R_3rd SOL ALIGN FPCB BW/FW PLS
MPUSH
AND       T4242	// R_3rd SS ALIGN FPCB FW
AND       T4245	// R_3rd SS ALIGN FPCB SUB BW
OUTP      M13842	// T)R_3rd SOL ALIGN FPCB BW >
MPOP
AND       T4243	// R_3rd SS ALIGN FPCB BW
OUTP      M13844	// T)R_3rd SOL ALIGN FPCB FW >
; L120
LOAD      M13906	// T)R_3rd SOL ALIGN FPCB SUB BW/FW
OUTP      M13850	// T)R_3rd SOL ALIGN FPCB SUB BW/FW PLS
; L121
LOAD      M13850	// T)R_3rd SOL ALIGN FPCB SUB BW/FW PLS
MPUSH
AND       T4244	// R_3rd SS ALIGN FPCB SUB FW
OUTP      M13852	// T)R_3rd SOL ALIGN FPCB SUB BW >
MPOP
AND       T4245	// R_3rd SS ALIGN FPCB SUB BW
AND       T4242	// R_3rd SS ALIGN FPCB FW
OUTP      M13854	// T)R_3rd SOL ALIGN FPCB SUB FW >
; L123
LOAD      M13908	// T)R_3rd SOL SUPPORT UP/DN
OUTP      M13860	// T)R_3rd SOL SUPPORT UP/DN PLS
; L124
LOAD      M13860	// T)R_3rd SOL SUPPORT UP/DN PLS
MPUSH
AND       T4247	// R_3rd SS SUPPORT UP
OUTP      M13862	// T)R_3rd SOL SUPPORT UP >
MPOP
AND       T4246	// R_3rd SS SUPPORT DN
OUTP      M13864	// T)R_3rd SOL SUPPORT DN >
// ======================== 4th TOOL ==========================
; L127
LOAD      M14400	// T)R_4th TOOL VC ON/OFF
OUTP      M14310	// T)4th_TOOL VC ON/OFF PLS

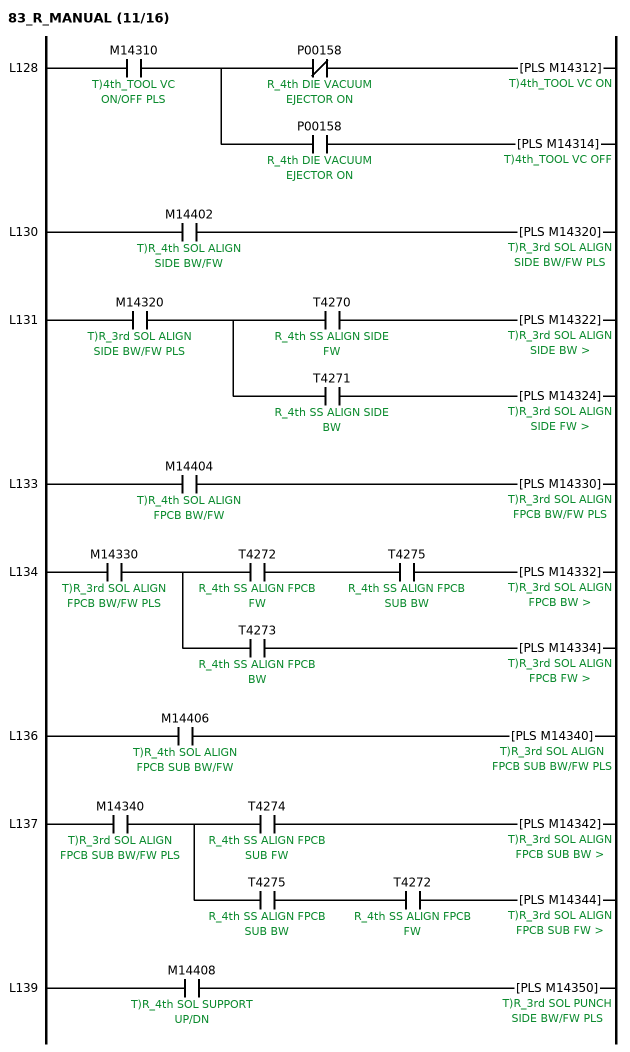
; L128
LOAD      M14310	// T)4th_TOOL VC ON/OFF PLS
MPUSH
AND NOT   P00158	// R_4th DIE VACUUM EJECTOR ON
OUTP      M14312	// T)4th_TOOL VC ON
MPOP
AND       P00158	// R_4th DIE VACUUM EJECTOR ON
OUTP      M14314	// T)4th_TOOL VC OFF
; L130
LOAD      M14402	// T)R_4th SOL ALIGN SIDE BW/FW
OUTP      M14320	// T)R_3rd SOL ALIGN SIDE BW/FW PLS
; L131
LOAD      M14320	// T)R_3rd SOL ALIGN SIDE BW/FW PLS
MPUSH
AND       T4270	// R_4th SS ALIGN SIDE FW
OUTP      M14322	// T)R_3rd SOL ALIGN SIDE BW >
MPOP
AND       T4271	// R_4th SS ALIGN SIDE BW
OUTP      M14324	// T)R_3rd SOL ALIGN SIDE FW >
; L133
LOAD      M14404	// T)R_4th SOL ALIGN FPCB BW/FW
OUTP      M14330	// T)R_3rd SOL ALIGN FPCB BW/FW PLS
; L134
LOAD      M14330	// T)R_3rd SOL ALIGN FPCB BW/FW PLS
MPUSH
AND       T4272	// R_4th SS ALIGN FPCB FW
AND       T4275	// R_4th SS ALIGN FPCB SUB BW
OUTP      M14332	// T)R_3rd SOL ALIGN FPCB BW >
MPOP
AND       T4273	// R_4th SS ALIGN FPCB BW
OUTP      M14334	// T)R_3rd SOL ALIGN FPCB FW >
; L136
LOAD      M14406	// T)R_4th SOL ALIGN FPCB SUB BW/FW
OUTP      M14340	// T)R_3rd SOL ALIGN FPCB SUB BW/FW PLS
; L137
LOAD      M14340	// T)R_3rd SOL ALIGN FPCB SUB BW/FW PLS
MPUSH
AND       T4274	// R_4th SS ALIGN FPCB SUB FW
OUTP      M14342	// T)R_3rd SOL ALIGN FPCB SUB BW >
MPOP
AND       T4275	// R_4th SS ALIGN FPCB SUB BW
AND       T4272	// R_4th SS ALIGN FPCB FW
OUTP      M14344	// T)R_3rd SOL ALIGN FPCB SUB FW >
; L139
LOAD      M14408	// T)R_4th SOL SUPPORT UP/DN
OUTP      M14350	// T)R_3rd SOL PUNCH SIDE BW/FW PLS

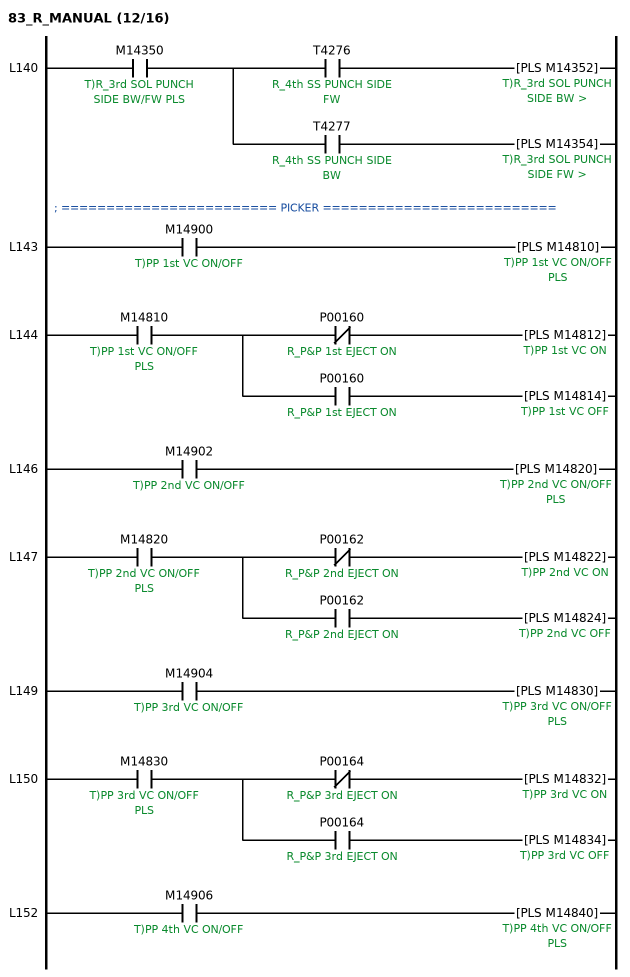
; L140
LOAD      M14350	// T)R_3rd SOL PUNCH SIDE BW/FW PLS
MPUSH
AND       T4276	// R_4th SS PUNCH SIDE FW
OUTP      M14352	// T)R_3rd SOL PUNCH SIDE BW >
MPOP
AND       T4277	// R_4th SS PUNCH SIDE BW
OUTP      M14354	// T)R_3rd SOL PUNCH SIDE FW >
// ======================== PICKER ==========================
; L143
LOAD      M14900	// T)PP 1st VC ON/OFF
OUTP      M14810	// T)PP 1st VC ON/OFF PLS
; L144
LOAD      M14810	// T)PP 1st VC ON/OFF PLS
MPUSH
AND NOT   P00160	// R_P&P 1st EJECT ON
OUTP      M14812	// T)PP 1st VC ON
MPOP
AND       P00160	// R_P&P 1st EJECT ON
OUTP      M14814	// T)PP 1st VC OFF
; L146
LOAD      M14902	// T)PP 2nd VC ON/OFF
OUTP      M14820	// T)PP 2nd VC ON/OFF PLS
; L147
LOAD      M14820	// T)PP 2nd VC ON/OFF PLS
MPUSH
AND NOT   P00162	// R_P&P 2nd EJECT ON
OUTP      M14822	// T)PP 2nd VC ON
MPOP
AND       P00162	// R_P&P 2nd EJECT ON
OUTP      M14824	// T)PP 2nd VC OFF
; L149
LOAD      M14904	// T)PP 3rd VC ON/OFF
OUTP      M14830	// T)PP 3rd VC ON/OFF PLS
; L150
LOAD      M14830	// T)PP 3rd VC ON/OFF PLS
MPUSH
AND NOT   P00164	// R_P&P 3rd EJECT ON
OUTP      M14832	// T)PP 3rd VC ON
MPOP
AND       P00164	// R_P&P 3rd EJECT ON
OUTP      M14834	// T)PP 3rd VC OFF
; L152
LOAD      M14906	// T)PP 4th VC ON/OFF
OUTP      M14840	// T)PP 4th VC ON/OFF PLS

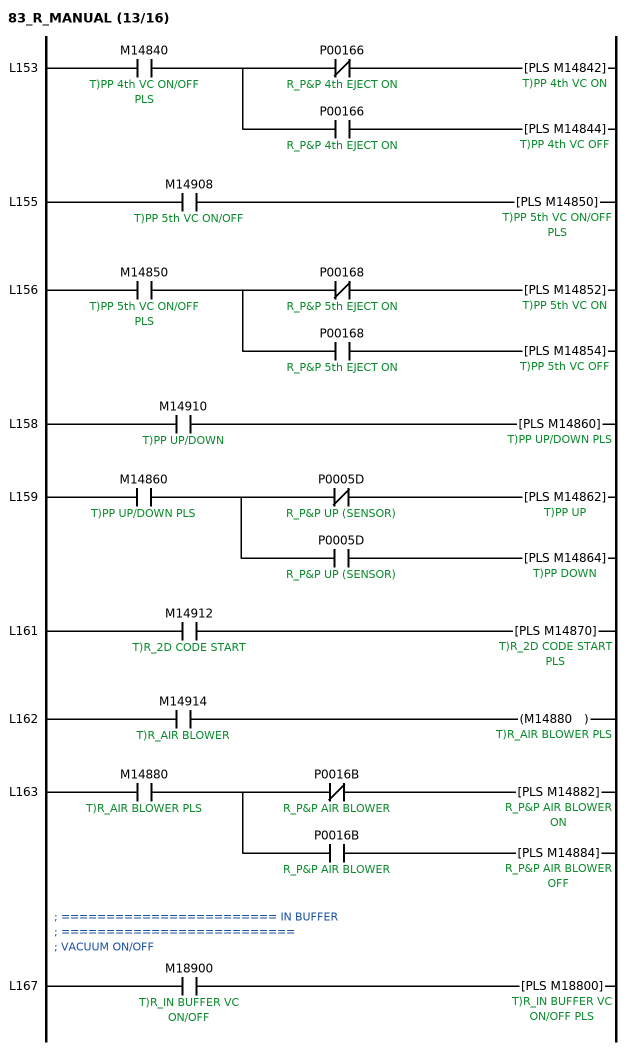
; L153
LOAD      M14840	// T)PP 4th VC ON/OFF PLS
MPUSH
AND NOT   P00166	// R_P&P 4th EJECT ON
OUTP      M14842	// T)PP 4th VC ON
MPOP
AND       P00166	// R_P&P 4th EJECT ON
OUTP      M14844	// T)PP 4th VC OFF
; L155
LOAD      M14908	// T)PP 5th VC ON/OFF
OUTP      M14850	// T)PP 5th VC ON/OFF PLS
; L156
LOAD      M14850	// T)PP 5th VC ON/OFF PLS
MPUSH
AND NOT   P00168	// R_P&P 5th EJECT ON
OUTP      M14852	// T)PP 5th VC ON
MPOP
AND       P00168	// R_P&P 5th EJECT ON
OUTP      M14854	// T)PP 5th VC OFF
; L158
LOAD      M14910	// T)PP UP/DOWN
OUTP      M14860	// T)PP UP/DOWN PLS
; L159
LOAD      M14860	// T)PP UP/DOWN PLS
MPUSH
AND NOT   P0005D	// R_P&P UP (SENSOR)
OUTP      M14862	// T)PP UP
MPOP
AND       P0005D	// R_P&P UP (SENSOR)
OUTP      M14864	// T)PP DOWN
; L161
LOAD      M14912	// T)R_2D CODE START
OUTP      M14870	// T)R_2D CODE START PLS
; L162
LOAD      M14914	// T)R_AIR BLOWER
OUT       M14880	// T)R_AIR BLOWER PLS
; L163
LOAD      M14880	// T)R_AIR BLOWER PLS
MPUSH
AND NOT   P0016B	// R_P&P AIR BLOWER
OUTP      M14882	// R_P&P AIR BLOWER ON
MPOP
AND       P0016B	// R_P&P AIR BLOWER
OUTP      M14884	// R_P&P AIR BLOWER OFF
// ======================== IN BUFFER ==========================
// VACUUM ON/OFF
; L167
LOAD      M18900	// T)R_IN BUFFER VC ON/OFF
OUTP      M18800	// T)R_IN BUFFER VC ON/OFF PLS

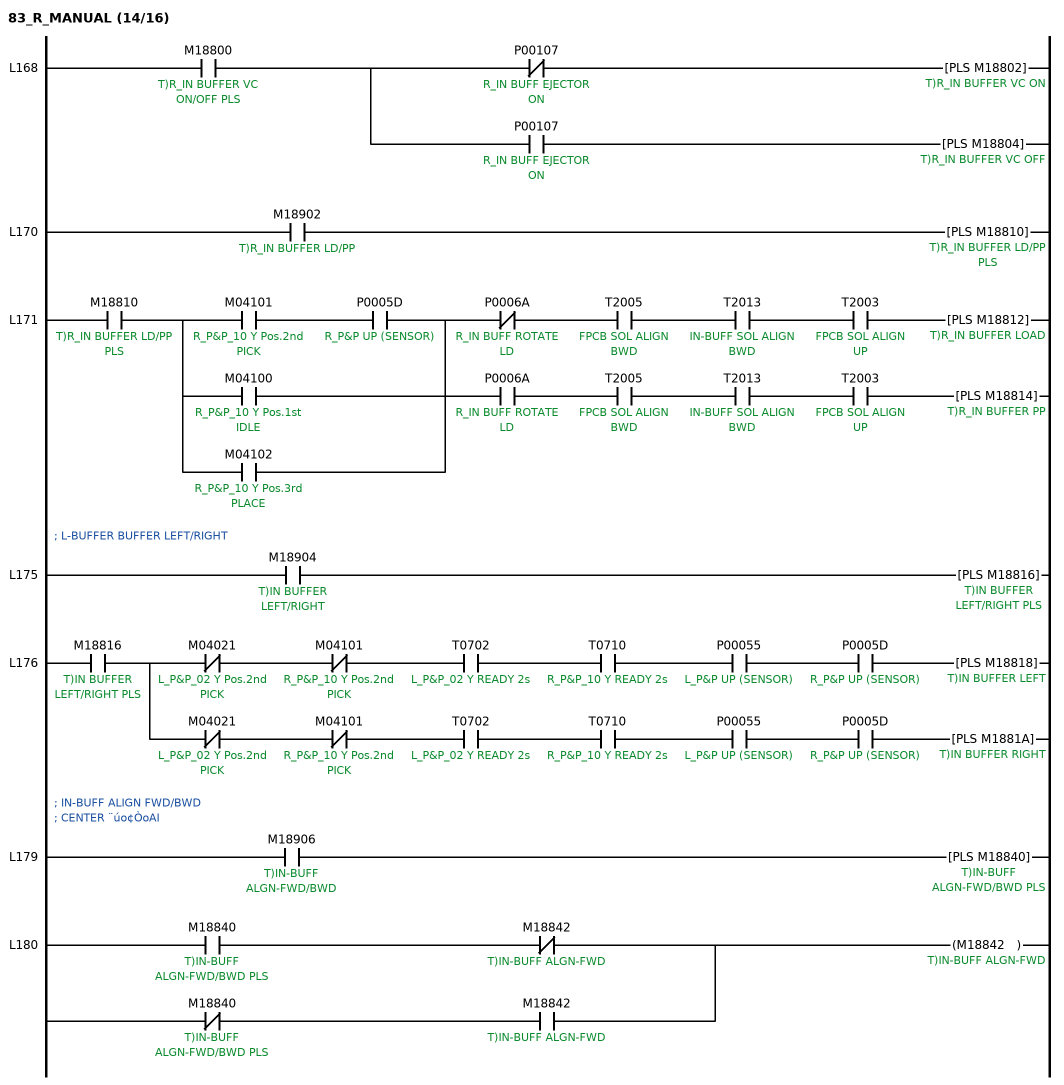
; L168
LOAD      M18800	// T)R_IN BUFFER VC ON/OFF PLS
MPUSH
AND NOT   P00107	// R_IN BUFF EJECTOR ON
OUTP      M18802	// T)R_IN BUFFER VC ON
MPOP
AND       P00107	// R_IN BUFF EJECTOR ON
OUTP      M18804	// T)R_IN BUFFER VC OFF
; L170
LOAD      M18902	// T)R_IN BUFFER LD/PP
OUTP      M18810	// T)R_IN BUFFER LD/PP PLS
; L171
LOAD      M18810	// T)R_IN BUFFER LD/PP PLS
LOAD      M04101	// R_P&P_10 Y Pos.2nd PICK
AND       P0005D	// R_P&P UP (SENSOR)
OR        M04100	// R_P&P_10 Y Pos.1st IDLE
OR        M04102	// R_P&P_10 Y Pos.3rd PLACE
AND LOAD
MPUSH
AND NOT   P0006A	// R_IN BUFF ROTATE      LD
AND       T2005	// FPCB SOL ALIGN         BWD
AND       T2013	// IN-BUFF SOL ALIGN BWD
AND       T2003	// FPCB SOL ALIGN         UP
OUTP      M18812	// T)R_IN BUFFER LOAD
MPOP
AND       P0006A	// R_IN BUFF ROTATE      LD
AND       T2005	// FPCB SOL ALIGN         BWD
AND       T2013	// IN-BUFF SOL ALIGN BWD
AND       T2003	// FPCB SOL ALIGN         UP
OUTP      M18814	// T)R_IN BUFFER PP
// L-BUFFER BUFFER LEFT/RIGHT
; L175
LOAD      M18904	// T)IN BUFFER LEFT/RIGHT
OUTP      M18816	// T)IN BUFFER LEFT/RIGHT PLS
; L176
LOAD      M18816	// T)IN BUFFER LEFT/RIGHT PLS
MPUSH
AND NOT   M04021	// L_P&P_02 Y Pos.2nd PICK
AND NOT   M04101	// R_P&P_10 Y Pos.2nd PICK
AND       T0702	// L_P&P_02 Y READY 2s
AND       T0710	// R_P&P_10 Y READY 2s
AND       P00055	// L_P&P UP (SENSOR)
AND       P0005D	// R_P&P UP (SENSOR)
OUTP      M18818	// T)IN BUFFER LEFT
MPOP
AND NOT   M04021	// L_P&P_02 Y Pos.2nd PICK
AND NOT   M04101	// R_P&P_10 Y Pos.2nd PICK
AND       T0702	// L_P&P_02 Y READY 2s
AND       T0710	// R_P&P_10 Y READY 2s
AND       P00055	// L_P&P UP (SENSOR)
AND       P0005D	// R_P&P UP (SENSOR)
OUTP      M1881A	// T)IN BUFFER RIGHT
// IN-BUFF ALIGN FWD/BWD
; L179
LOAD      M18906	// T)IN-BUFF ALGN-FWD/BWD
OUTP      M18840	// T)IN-BUFF ALGN-FWD/BWD PLS
// output comment: CENTER ¨úo¢ÒoAI
; L180
LOAD      M18840	// T)IN-BUFF ALGN-FWD/BWD PLS
AND NOT   M18842	// T)IN-BUFF ALGN-FWD
LOAD NOT  M18840	// T)IN-BUFF ALGN-FWD/BWD PLS
AND       M18842	// T)IN-BUFF ALGN-FWD
OR LOAD
OUT       M18842	// T)IN-BUFF ALGN-FWD

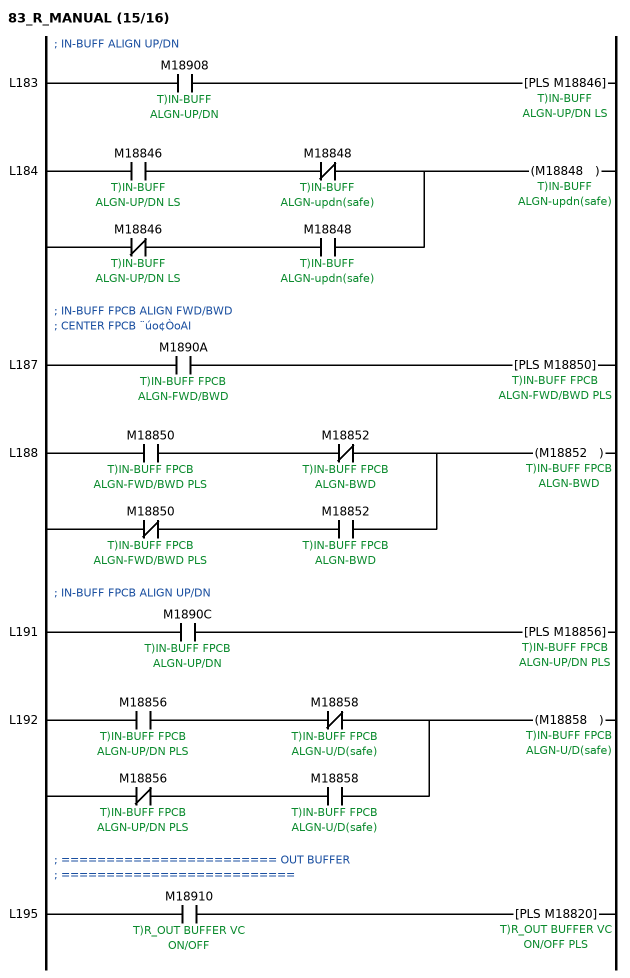
// IN-BUFF ALIGN UP/DN
; L183
LOAD      M18908	// T)IN-BUFF ALGN-UP/DN
OUTP      M18846	// T)IN-BUFF ALGN-UP/DN LS
; L184
LOAD      M18846	// T)IN-BUFF ALGN-UP/DN LS
AND NOT   M18848	// T)IN-BUFF ALGN-updn(safe)
LOAD NOT  M18846	// T)IN-BUFF ALGN-UP/DN LS
AND       M18848	// T)IN-BUFF ALGN-updn(safe)
OR LOAD
OUT       M18848	// T)IN-BUFF ALGN-updn(safe)
// IN-BUFF FPCB ALIGN FWD/BWD
; L187
LOAD      M1890A	// T)IN-BUFF FPCB ALGN-FWD/BWD
OUTP      M18850	// T)IN-BUFF FPCB ALGN-FWD/BWD PLS
// output comment: CENTER FPCB ¨úo¢ÒoAI
; L188
LOAD      M18850	// T)IN-BUFF FPCB ALGN-FWD/BWD PLS
AND NOT   M18852	// T)IN-BUFF FPCB ALGN-BWD
LOAD NOT  M18850	// T)IN-BUFF FPCB ALGN-FWD/BWD PLS
AND       M18852	// T)IN-BUFF FPCB ALGN-BWD
OR LOAD
OUT       M18852	// T)IN-BUFF FPCB ALGN-BWD
// IN-BUFF FPCB ALIGN UP/DN
; L191
LOAD      M1890C	// T)IN-BUFF FPCB ALGN-UP/DN
OUTP      M18856	// T)IN-BUFF FPCB ALGN-UP/DN PLS
; L192
LOAD      M18856	// T)IN-BUFF FPCB ALGN-UP/DN PLS
AND NOT   M18858	// T)IN-BUFF FPCB ALGN-U/D(safe)
LOAD NOT  M18856	// T)IN-BUFF FPCB ALGN-UP/DN PLS
AND       M18858	// T)IN-BUFF FPCB ALGN-U/D(safe)
OR LOAD
OUT       M18858	// T)IN-BUFF FPCB ALGN-U/D(safe)
// ======================== OUT BUFFER ==========================
; L195
LOAD      M18910	// T)R_OUT BUFFER VC ON/OFF
OUTP      M18820	// T)R_OUT BUFFER VC ON/OFF PLS

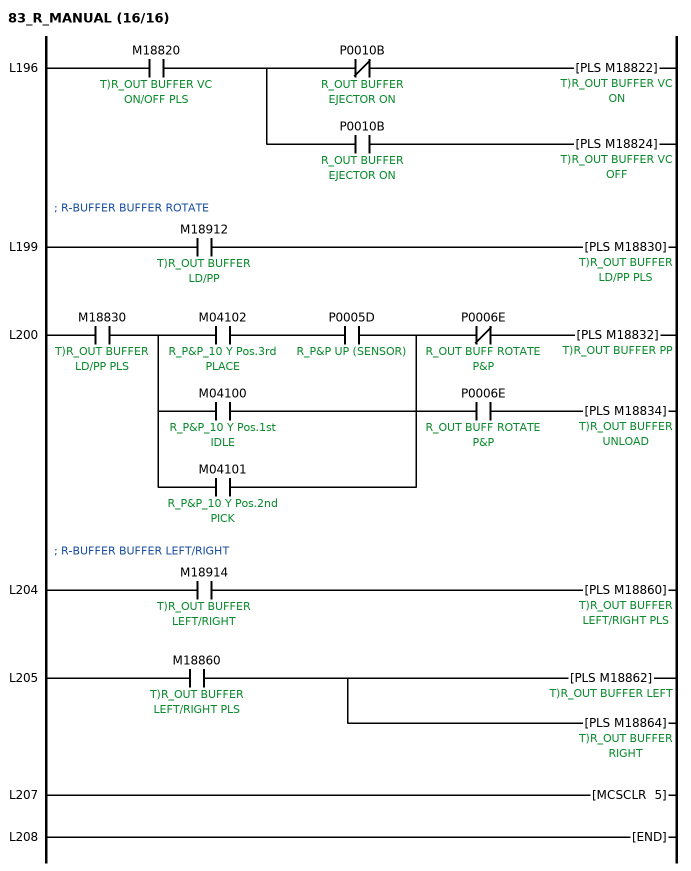
; L196
LOAD      M18820	// T)R_OUT BUFFER VC ON/OFF PLS
MPUSH
AND NOT   P0010B	// R_OUT BUFFER EJECTOR ON
OUTP      M18822	// T)R_OUT BUFFER VC ON
MPOP
AND       P0010B	// R_OUT BUFFER EJECTOR ON
OUTP      M18824	// T)R_OUT BUFFER VC OFF
// R-BUFFER BUFFER ROTATE
; L199
LOAD      M18912	// T)R_OUT BUFFER LD/PP
OUTP      M18830	// T)R_OUT BUFFER LD/PP PLS
; L200
LOAD      M18830	// T)R_OUT BUFFER LD/PP PLS
LOAD      M04102	// R_P&P_10 Y Pos.3rd PLACE
AND       P0005D	// R_P&P UP (SENSOR)
OR        M04100	// R_P&P_10 Y Pos.1st IDLE
OR        M04101	// R_P&P_10 Y Pos.2nd PICK
AND LOAD
MPUSH
AND NOT   P0006E	// R_OUT BUFF ROTATE      P&P
OUTP      M18832	// T)R_OUT BUFFER PP
MPOP
AND       P0006E	// R_OUT BUFF ROTATE      P&P
OUTP      M18834	// T)R_OUT BUFFER UNLOAD
// R-BUFFER BUFFER LEFT/RIGHT
; L204
LOAD      M18914	// T)R_OUT BUFFER LEFT/RIGHT
OUTP      M18860	// T)R_OUT BUFFER LEFT/RIGHT PLS
; L205
LOAD      M18860	// T)R_OUT BUFFER LEFT/RIGHT PLS
OUTP      M18862	// T)R_OUT BUFFER LEFT
OUTP      M18864	// T)R_OUT BUFFER RIGHT
; L207
MCSCLR    5
; L208
END

PROGRAM 84_RUN_TIME (task: ¨ö¨¬A¥ì CA¡¤I¡¾¡¿¡¤¡Í)

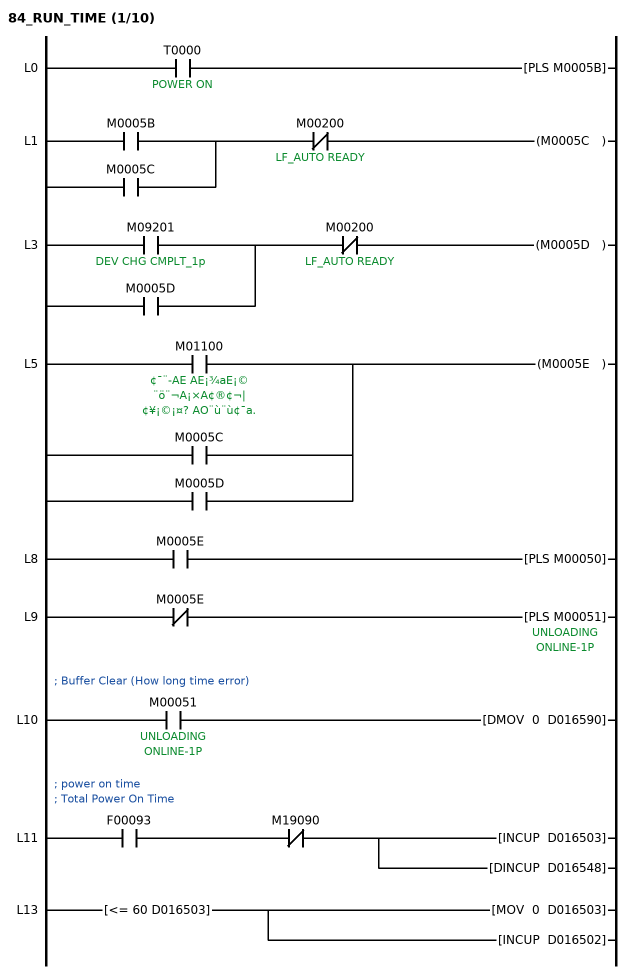
; L0
LOAD      T0000	// POWER ON
OUTP      M0005B
; L1
LOAD      M0005B
OR        M0005C
AND NOT   M00200	// LF_AUTO READY
OUT       M0005C
; L3
LOAD      M09201	// DEV CHG CMPLT_1p
OR        M0005D
AND NOT   M00200	// LF_AUTO READY
OUT       M0005D
; L5
LOAD      M01100	// ¢¯¨­AE AE¡¾aE¡© ¨ö¨¬A¡×A¢®¢¬| ¢¥¡©¡¤? AO¨ù¨ù¢¯a.
OR        M0005C
OR        M0005D
OUT       M0005E
; L8
LOAD      M0005E
OUTP      M00050
; L9
LOAD NOT  M0005E
OUTP      M00051	// UNLOADING ONLINE-1P
; L10
LOAD      M00051	// UNLOADING ONLINE-1P
DMOV      0 D016590
// output comment: Buffer Clear (How long time error)
; L11
LOAD      F00093
AND NOT   M19090
INCUP     D016503
DINCUP    D016548
// output comment: power on time
// output comment: Total Power On Time
; L13
LOAD<=    60 D016503
MOV       0 D016503
INCUP     D016502

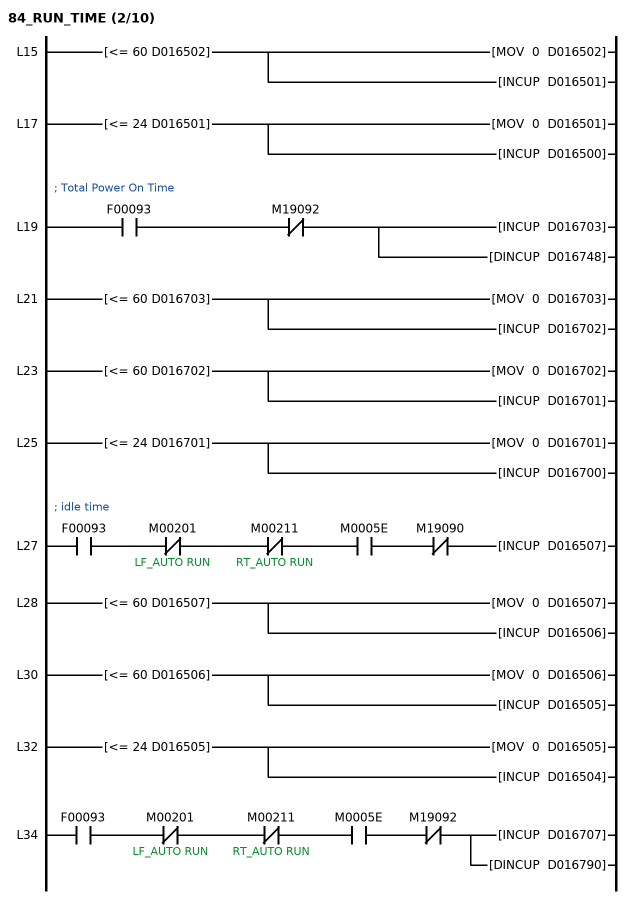
; L15
LOAD<=    60 D016502
MOV       0 D016502
INCUP     D016501
; L17
LOAD<=    24 D016501
MOV       0 D016501
INCUP     D016500
; L19
LOAD      F00093
AND NOT   M19092
INCUP     D016703
DINCUP    D016748
// output comment: Total Power On Time
; L21
LOAD<=    60 D016703
MOV       0 D016703
INCUP     D016702
; L23
LOAD<=    60 D016702
MOV       0 D016702
INCUP     D016701
; L25
LOAD<=    24 D016701
MOV       0 D016701
INCUP     D016700
; L27
LOAD      F00093
AND NOT   M00201	// LF_AUTO RUN
AND NOT   M00211	// RT_AUTO RUN
AND       M0005E
AND NOT   M19090
INCUP     D016507
// output comment: idle time
; L28
LOAD<=    60 D016507
MOV       0 D016507
INCUP     D016506
; L30
LOAD<=    60 D016506
MOV       0 D016506
INCUP     D016505
; L32
LOAD<=    24 D016505
MOV       0 D016505
INCUP     D016504
; L34
LOAD      F00093
AND NOT   M00201	// LF_AUTO RUN
AND NOT   M00211	// RT_AUTO RUN
AND       M0005E
AND NOT   M19092
INCUP     D016707
DINCUP    D016790

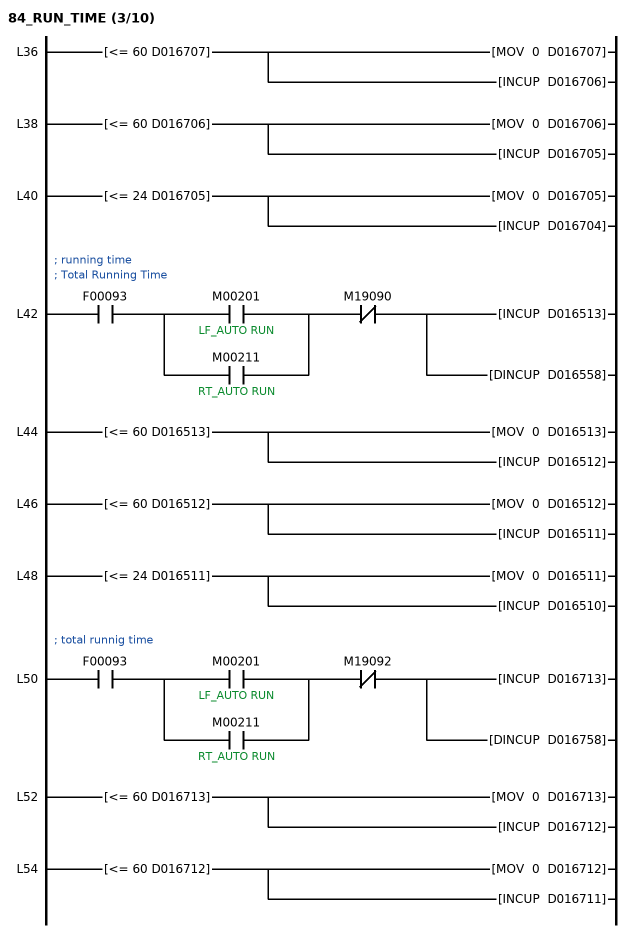
; L36
LOAD<=    60 D016707
MOV       0 D016707
INCUP     D016706
; L38
LOAD<=    60 D016706
MOV       0 D016706
INCUP     D016705
; L40
LOAD<=    24 D016705
MOV       0 D016705
INCUP     D016704
; L42
LOAD      F00093
LOAD      M00201	// LF_AUTO RUN
OR        M00211	// RT_AUTO RUN
AND LOAD
AND NOT   M19090
INCUP     D016513
DINCUP    D016558
// output comment: running time
// output comment: Total Running Time
; L44
LOAD<=    60 D016513
MOV       0 D016513
INCUP     D016512
; L46
LOAD<=    60 D016512
MOV       0 D016512
INCUP     D016511
; L48
LOAD<=    24 D016511
MOV       0 D016511
INCUP     D016510
; L50
LOAD      F00093
LOAD      M00201	// LF_AUTO RUN
OR        M00211	// RT_AUTO RUN
AND LOAD
AND NOT   M19092
INCUP     D016713
DINCUP    D016758
// output comment: total runnig time
; L52
LOAD<=    60 D016713
MOV       0 D016713
INCUP     D016712
; L54
LOAD<=    60 D016712
MOV       0 D016712
INCUP     D016711

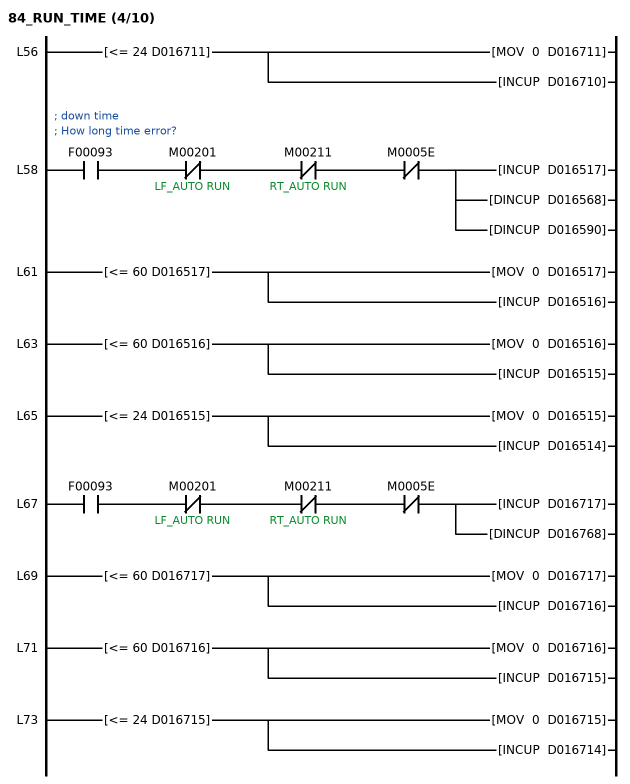
; L56
LOAD<=    24 D016711
MOV       0 D016711
INCUP     D016710
; L58
LOAD      F00093
AND NOT   M00201	// LF_AUTO RUN
AND NOT   M00211	// RT_AUTO RUN
AND NOT   M0005E
INCUP     D016517
DINCUP    D016568
DINCUP    D016590
// output comment: down time
// output comment: How long time error?
; L61
LOAD<=    60 D016517
MOV       0 D016517
INCUP     D016516
; L63
LOAD<=    60 D016516
MOV       0 D016516
INCUP     D016515
; L65
LOAD<=    24 D016515
MOV       0 D016515
INCUP     D016514
; L67
LOAD      F00093
AND NOT   M00201	// LF_AUTO RUN
AND NOT   M00211	// RT_AUTO RUN
AND NOT   M0005E
INCUP     D016717
DINCUP    D016768
; L69
LOAD<=    60 D016717
MOV       0 D016717
INCUP     D016716
; L71
LOAD<=    60 D016716
MOV       0 D016716
INCUP     D016715
; L73
LOAD<=    24 D016715
MOV       0 D016715
INCUP     D016714

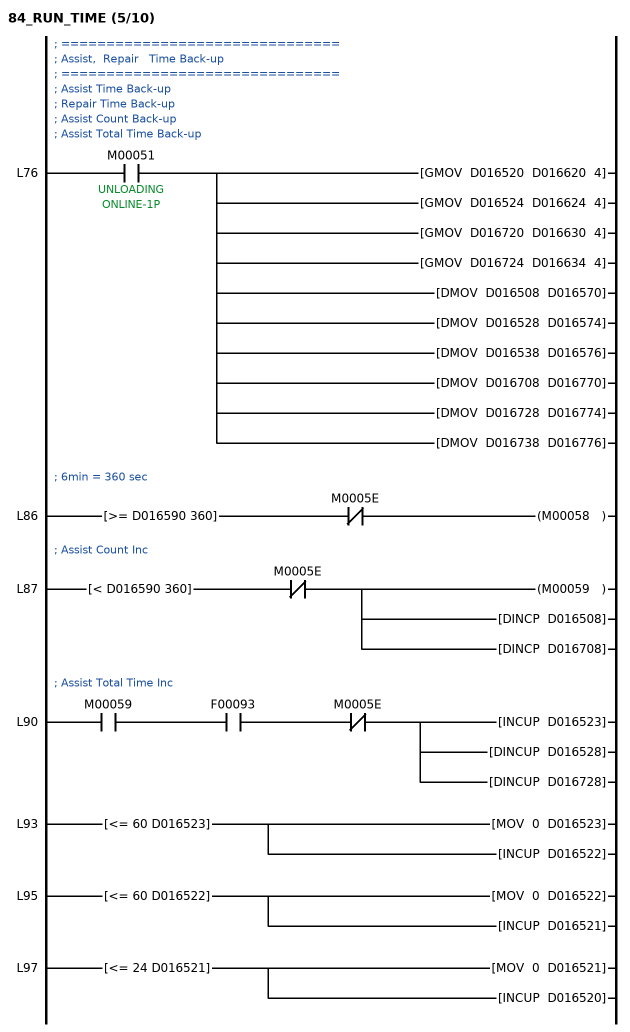
// ===============================
// Assist,  Repair   Time Back-up
// ===============================
; L76
LOAD      M00051	// UNLOADING ONLINE-1P
GMOV      D016520 D016620 4
GMOV      D016524 D016624 4
GMOV      D016720 D016630 4
GMOV      D016724 D016634 4
DMOV      D016508 D016570
DMOV      D016528 D016574
DMOV      D016538 D016576
DMOV      D016708 D016770
DMOV      D016728 D016774
DMOV      D016738 D016776
// output comment: Assist Time Back-up
// output comment: Repair Time Back-up
// output comment: Assist Count Back-up
// output comment: Assist Total Time Back-up
; L86
LOAD>=    D016590 360
AND NOT   M0005E
OUT       M00058
// output comment: 6min = 360 sec
; L87
LOAD<     D016590 360
AND NOT   M0005E
OUT       M00059
DINCP     D016508
DINCP     D016708
// output comment: Assist Count Inc
; L90
LOAD      M00059
AND       F00093
AND NOT   M0005E
INCUP     D016523
DINCUP    D016528
DINCUP    D016728
// output comment: Assist Total Time Inc
; L93
LOAD<=    60 D016523
MOV       0 D016523
INCUP     D016522
; L95
LOAD<=    60 D016522
MOV       0 D016522
INCUP     D016521
; L97
LOAD<=    24 D016521
MOV       0 D016521
INCUP     D016520

